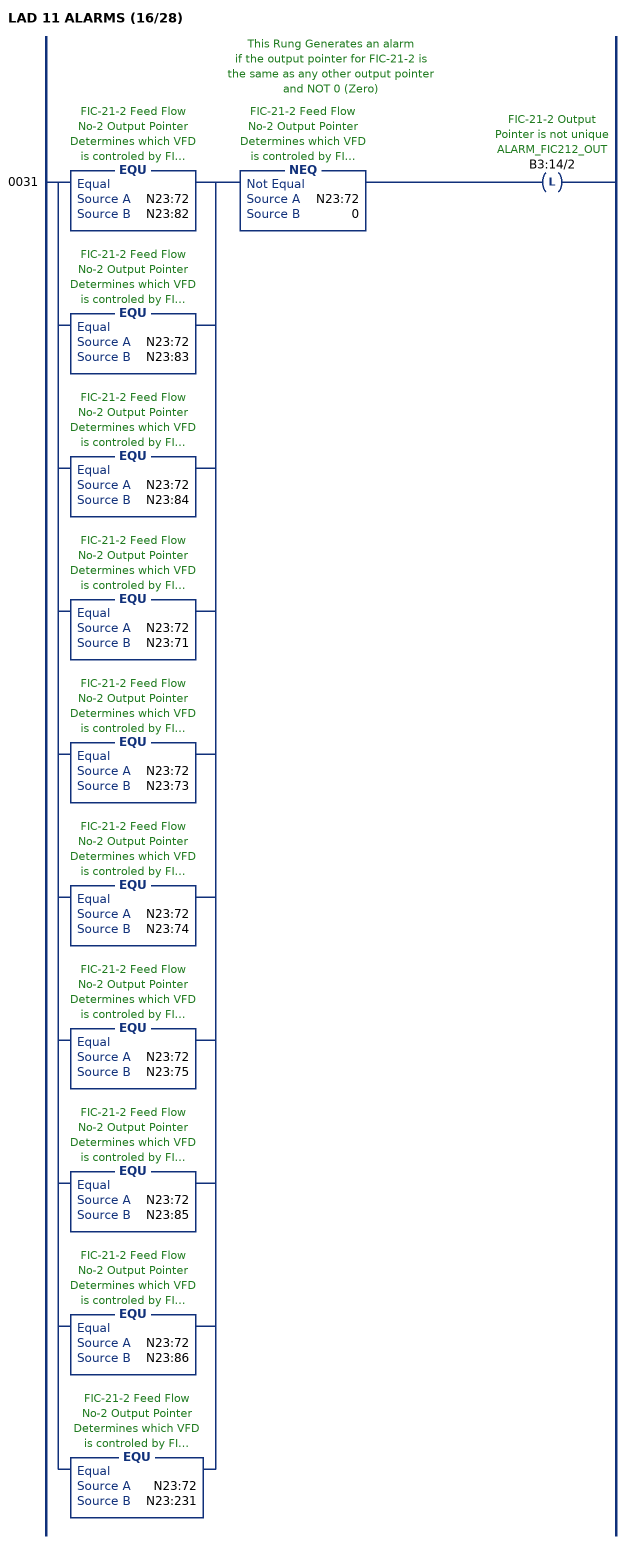
% Rung: 31 %
% This Rung Generates an alarm
% if the output pointer for FIC-21-2 is
% the same as any other output pointer
% and NOT 0 (Zero) %
SOR BST EQU N23:72 N23:82 NXB EQU N23:72 N23:83 NXB EQU N23:72 N23:84 NXB EQU N23:72 N23:71 NXB EQU N23:72 N23:73 NXB EQU N23:72 N23:74 NXB EQU N23:72 N23:75 NXB EQU N23:72 N23:85 NXB EQU N23:72 N23:86 NXB EQU N23:72 N23:231 BND NEQ N23:72 0 OTL B3:14/2 EOR
%   N23:72  FIC212_OUT_PTR  "FIC-21-2 Feed Flow No-2 Output Pointer Determines which VFD is controled by FIC" %
%   N23:82  EV02_OUT_PTR  "EV-2 Rotor Output Pointer (Selects which VFD is used by EV-2)" %
%   N23:83  EV03_OUT_PTR  "EV-3 Rotor Drive Output Pointer (Selects which VFD is used by EV-3)" %
%   N23:84  AG04_OUT_PTR  "AG-4 Agitator Output Pointer (Selects which VFD is used by AG-4)" %
%   N23:71  FIC211_OUT_PTR  "FIC-21-1 Feed Flow No-1 Output Pointer Determines which VFD is controled by FIC" %
%   N23:73  FIC213_OUT_PTR  "FIC-21-3 Feed Flow No-3 Output Pointer Determines which VFD is controled by FIC" %
%   N23:74  FIC214_OUT_PTR  "FIC-21-4 Feed Flow No-4 Output Pointer Determines which VFD is controled by FIC" %
%   N23:75  PIC461_OUT_PTR  "PIC-46-1 Flash Evap Feed Pres Output Pointer Determines which VFD is controled by FIC" %
%   N23:85  EV42_OUT_PTR  "EV-42 Rotor Drive Rotor Output Pointer (Selects which VFD is used by EV-3)" %
%   N23:86  EV20_OUT_PTR  "EV-20 Rotor Drive Rotor Output Pointer (Selects which VFD is used by EV-3)" %
%   N23:231  LIC221_OUT_PTR  "LIC-22-1 Level No-1 Output Pointer Determines which VFD is controled by LIC" %
%   B3:14/2  ALARM_FIC212_OUT  "FIC-21-2 Output Pointer is not unique" %

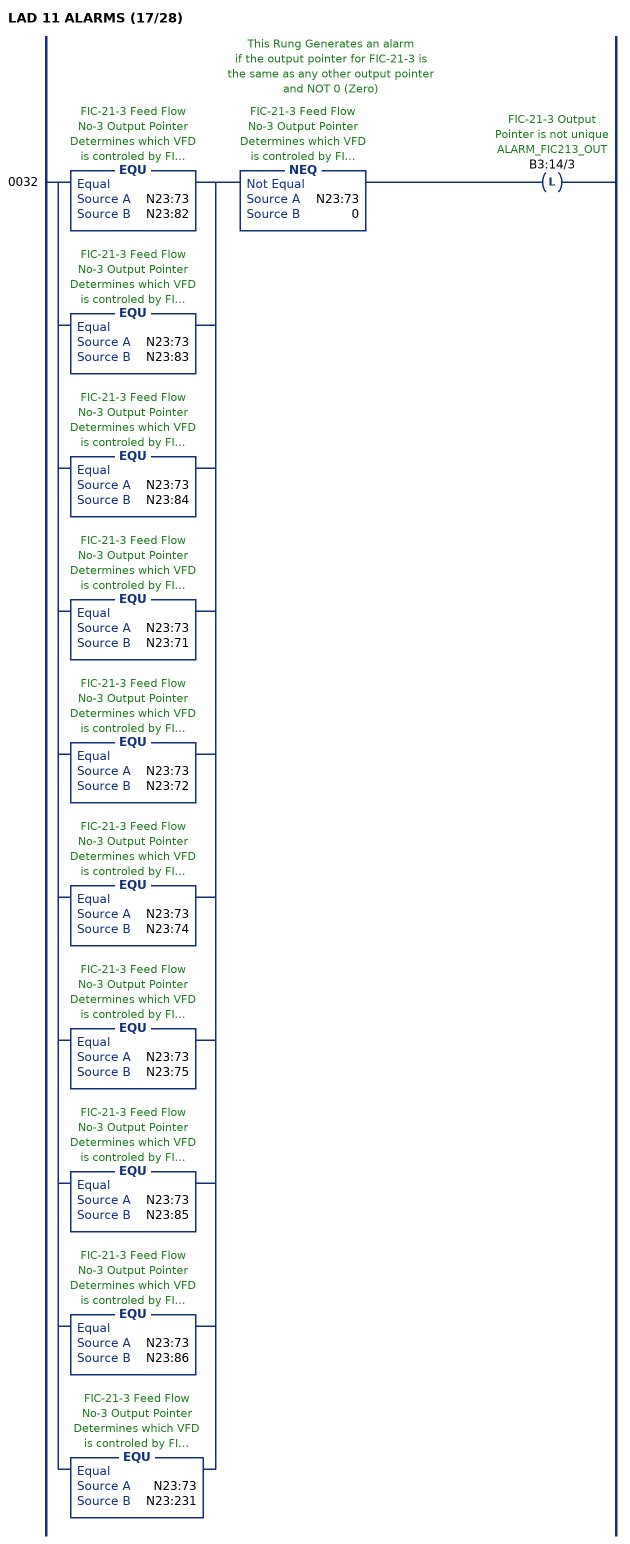
% Rung: 32 %
% This Rung Generates an alarm
% if the output pointer for FIC-21-3 is
% the same as any other output pointer
% and NOT 0 (Zero) %
SOR BST EQU N23:73 N23:82 NXB EQU N23:73 N23:83 NXB EQU N23:73 N23:84 NXB EQU N23:73 N23:71 NXB EQU N23:73 N23:72 NXB EQU N23:73 N23:74 NXB EQU N23:73 N23:75 NXB EQU N23:73 N23:85 NXB EQU N23:73 N23:86 NXB EQU N23:73 N23:231 BND NEQ N23:73 0 OTL B3:14/3 EOR
%   N23:73  FIC213_OUT_PTR  "FIC-21-3 Feed Flow No-3 Output Pointer Determines which VFD is controled by FIC" %
%   N23:82  EV02_OUT_PTR  "EV-2 Rotor Output Pointer (Selects which VFD is used by EV-2)" %
%   N23:83  EV03_OUT_PTR  "EV-3 Rotor Drive Output Pointer (Selects which VFD is used by EV-3)" %
%   N23:84  AG04_OUT_PTR  "AG-4 Agitator Output Pointer (Selects which VFD is used by AG-4)" %
%   N23:71  FIC211_OUT_PTR  "FIC-21-1 Feed Flow No-1 Output Pointer Determines which VFD is controled by FIC" %
%   N23:72  FIC212_OUT_PTR  "FIC-21-2 Feed Flow No-2 Output Pointer Determines which VFD is controled by FIC" %
%   N23:74  FIC214_OUT_PTR  "FIC-21-4 Feed Flow No-4 Output Pointer Determines which VFD is controled by FIC" %
%   N23:75  PIC461_OUT_PTR  "PIC-46-1 Flash Evap Feed Pres Output Pointer Determines which VFD is controled by FIC" %
%   N23:85  EV42_OUT_PTR  "EV-42 Rotor Drive Rotor Output Pointer (Selects which VFD is used by EV-3)" %
%   N23:86  EV20_OUT_PTR  "EV-20 Rotor Drive Rotor Output Pointer (Selects which VFD is used by EV-3)" %
%   N23:231  LIC221_OUT_PTR  "LIC-22-1 Level No-1 Output Pointer Determines which VFD is controled by LIC" %
%   B3:14/3  ALARM_FIC213_OUT  "FIC-21-3 Output Pointer is not unique" %

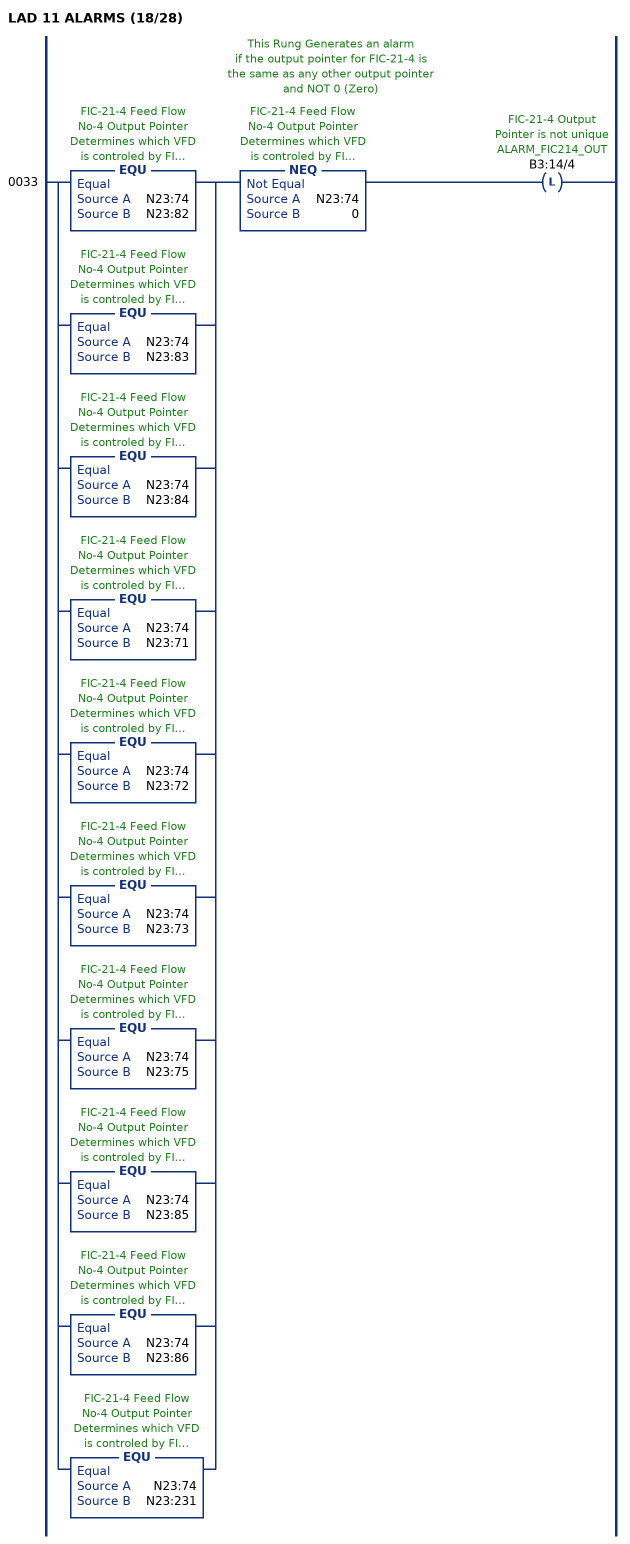
% Rung: 33 %
% This Rung Generates an alarm
% if the output pointer for FIC-21-4 is
% the same as any other output pointer
% and NOT 0 (Zero) %
SOR BST EQU N23:74 N23:82 NXB EQU N23:74 N23:83 NXB EQU N23:74 N23:84 NXB EQU N23:74 N23:71 NXB EQU N23:74 N23:72 NXB EQU N23:74 N23:73 NXB EQU N23:74 N23:75 NXB EQU N23:74 N23:85 NXB EQU N23:74 N23:86 NXB EQU N23:74 N23:231 BND NEQ N23:74 0 OTL B3:14/4 EOR
%   N23:74  FIC214_OUT_PTR  "FIC-21-4 Feed Flow No-4 Output Pointer Determines which VFD is controled by FIC" %
%   N23:82  EV02_OUT_PTR  "EV-2 Rotor Output Pointer (Selects which VFD is used by EV-2)" %
%   N23:83  EV03_OUT_PTR  "EV-3 Rotor Drive Output Pointer (Selects which VFD is used by EV-3)" %
%   N23:84  AG04_OUT_PTR  "AG-4 Agitator Output Pointer (Selects which VFD is used by AG-4)" %
%   N23:71  FIC211_OUT_PTR  "FIC-21-1 Feed Flow No-1 Output Pointer Determines which VFD is controled by FIC" %
%   N23:72  FIC212_OUT_PTR  "FIC-21-2 Feed Flow No-2 Output Pointer Determines which VFD is controled by FIC" %
%   N23:73  FIC213_OUT_PTR  "FIC-21-3 Feed Flow No-3 Output Pointer Determines which VFD is controled by FIC" %
%   N23:75  PIC461_OUT_PTR  "PIC-46-1 Flash Evap Feed Pres Output Pointer Determines which VFD is controled by FIC" %
%   N23:85  EV42_OUT_PTR  "EV-42 Rotor Drive Rotor Output Pointer (Selects which VFD is used by EV-3)" %
%   N23:86  EV20_OUT_PTR  "EV-20 Rotor Drive Rotor Output Pointer (Selects which VFD is used by EV-3)" %
%   N23:231  LIC221_OUT_PTR  "LIC-22-1 Level No-1 Output Pointer Determines which VFD is controled by LIC" %
%   B3:14/4  ALARM_FIC214_OUT  "FIC-21-4 Output Pointer is not unique" %

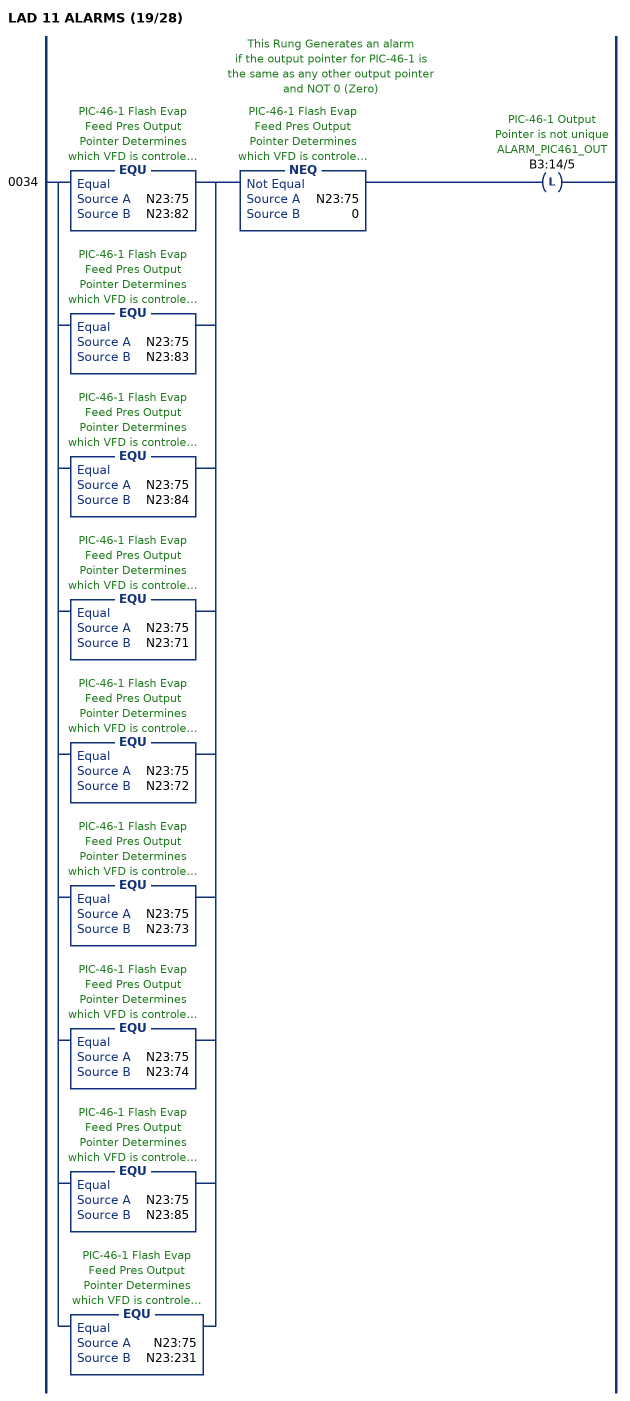
% Rung: 34 %
% This Rung Generates an alarm
% if the output pointer for PIC-46-1 is
% the same as any other output pointer
% and NOT 0 (Zero) %
SOR BST EQU N23:75 N23:82 NXB EQU N23:75 N23:83 NXB EQU N23:75 N23:84 NXB EQU N23:75 N23:71 NXB EQU N23:75 N23:72 NXB EQU N23:75 N23:73 NXB EQU N23:75 N23:74 NXB EQU N23:75 N23:85 NXB EQU N23:75 N23:231 BND NEQ N23:75 0 OTL B3:14/5 EOR
%   N23:75  PIC461_OUT_PTR  "PIC-46-1 Flash Evap Feed Pres Output Pointer Determines which VFD is controled by FIC" %
%   N23:82  EV02_OUT_PTR  "EV-2 Rotor Output Pointer (Selects which VFD is used by EV-2)" %
%   N23:83  EV03_OUT_PTR  "EV-3 Rotor Drive Output Pointer (Selects which VFD is used by EV-3)" %
%   N23:84  AG04_OUT_PTR  "AG-4 Agitator Output Pointer (Selects which VFD is used by AG-4)" %
%   N23:71  FIC211_OUT_PTR  "FIC-21-1 Feed Flow No-1 Output Pointer Determines which VFD is controled by FIC" %
%   N23:72  FIC212_OUT_PTR  "FIC-21-2 Feed Flow No-2 Output Pointer Determines which VFD is controled by FIC" %
%   N23:73  FIC213_OUT_PTR  "FIC-21-3 Feed Flow No-3 Output Pointer Determines which VFD is controled by FIC" %
%   N23:74  FIC214_OUT_PTR  "FIC-21-4 Feed Flow No-4 Output Pointer Determines which VFD is controled by FIC" %
%   N23:85  EV42_OUT_PTR  "EV-42 Rotor Drive Rotor Output Pointer (Selects which VFD is used by EV-3)" %
%   N23:231  LIC221_OUT_PTR  "LIC-22-1 Level No-1 Output Pointer Determines which VFD is controled by LIC" %
%   B3:14/5  ALARM_PIC461_OUT  "PIC-46-1 Output Pointer is not unique" %

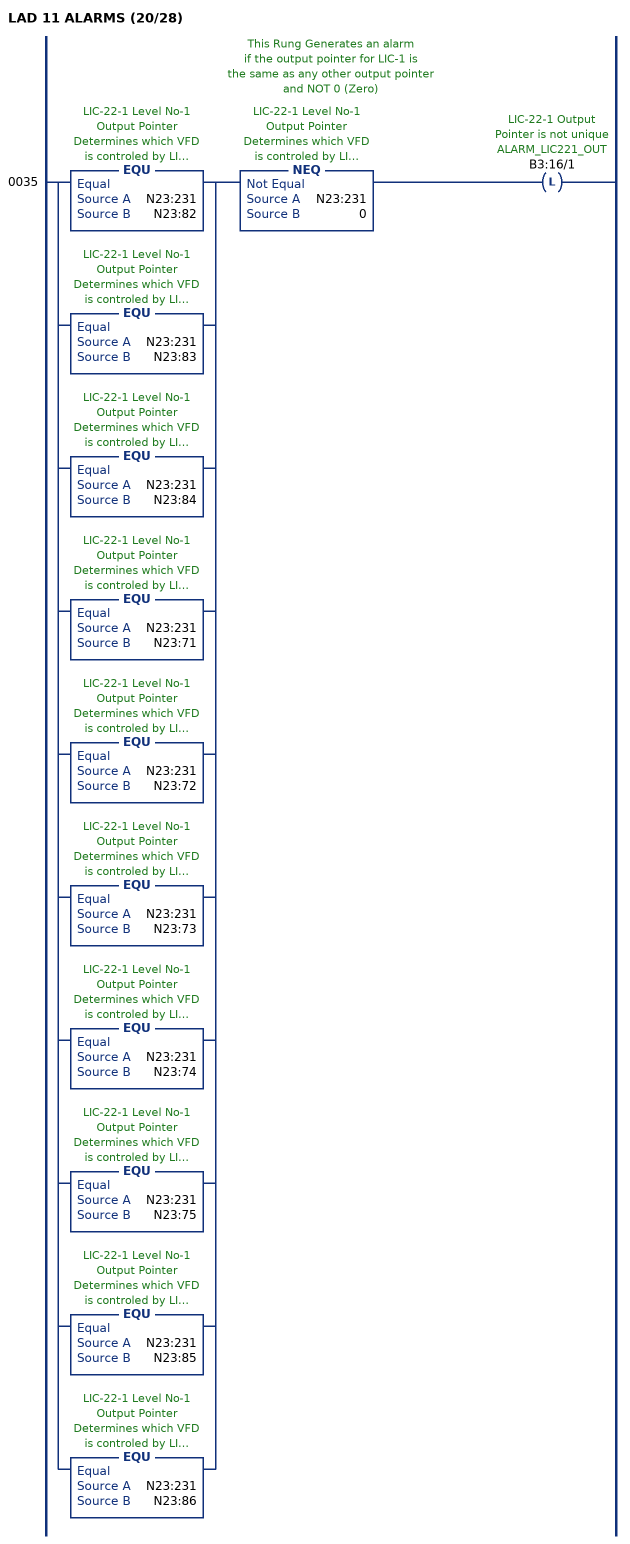
% Rung: 35 %
% This Rung Generates an alarm
% if the output pointer for LIC-1 is
% the same as any other output pointer
% and NOT 0 (Zero) %
SOR BST EQU N23:231 N23:82 NXB EQU N23:231 N23:83 NXB EQU N23:231 N23:84 NXB EQU N23:231 N23:71 NXB EQU N23:231 N23:72 NXB EQU N23:231 N23:73 NXB EQU N23:231 N23:74 NXB EQU N23:231 N23:75 NXB EQU N23:231 N23:85 NXB EQU N23:231 N23:86 BND NEQ N23:231 0 OTL B3:16/1 EOR
%   N23:231  LIC221_OUT_PTR  "LIC-22-1 Level No-1 Output Pointer Determines which VFD is controled by LIC" %
%   N23:82  EV02_OUT_PTR  "EV-2 Rotor Output Pointer (Selects which VFD is used by EV-2)" %
%   N23:83  EV03_OUT_PTR  "EV-3 Rotor Drive Output Pointer (Selects which VFD is used by EV-3)" %
%   N23:84  AG04_OUT_PTR  "AG-4 Agitator Output Pointer (Selects which VFD is used by AG-4)" %
%   N23:71  FIC211_OUT_PTR  "FIC-21-1 Feed Flow No-1 Output Pointer Determines which VFD is controled by FIC" %
%   N23:72  FIC212_OUT_PTR  "FIC-21-2 Feed Flow No-2 Output Pointer Determines which VFD is controled by FIC" %
%   N23:73  FIC213_OUT_PTR  "FIC-21-3 Feed Flow No-3 Output Pointer Determines which VFD is controled by FIC" %
%   N23:74  FIC214_OUT_PTR  "FIC-21-4 Feed Flow No-4 Output Pointer Determines which VFD is controled by FIC" %
%   N23:75  PIC461_OUT_PTR  "PIC-46-1 Flash Evap Feed Pres Output Pointer Determines which VFD is controled by FIC" %
%   N23:85  EV42_OUT_PTR  "EV-42 Rotor Drive Rotor Output Pointer (Selects which VFD is used by EV-3)" %
%   N23:86  EV20_OUT_PTR  "EV-20 Rotor Drive Rotor Output Pointer (Selects which VFD is used by EV-3)" %
%   B3:16/1  ALARM_LIC221_OUT  "LIC-22-1 Output Pointer is not unique" %

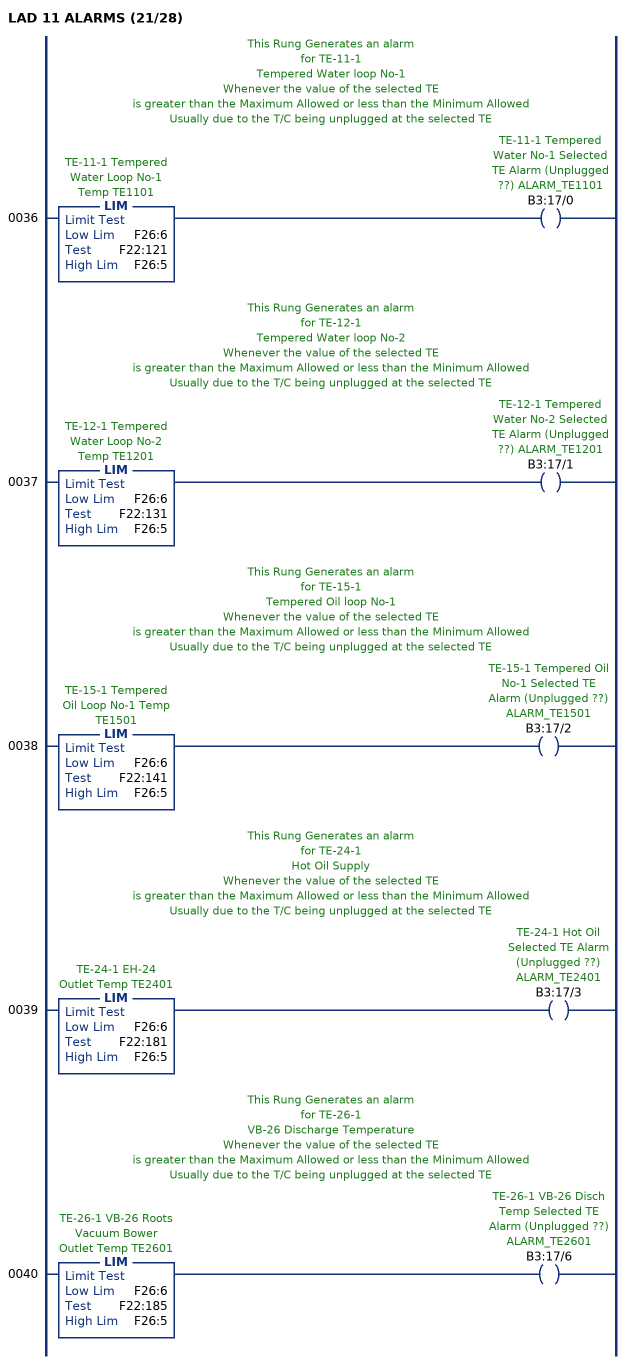
% Rung: 36 %
% This Rung Generates an alarm
% for TE-11-1
% Tempered Water loop No-1
% Whenever the value of the selected TE
% is greater than the Maximum Allowed or less than the Minimum Allowed
% Usually due to the T/C being unplugged at the selected TE %
SOR LIM F26:6 F22:121 F26:5 OTE B3:17/0 EOR
%   F26:6  TE_MAX  "TE Input Maximum Value if TE is >= this value an alarm is generated" %
%   F22:121  TE1101  "TE-11-1 Tempered Water Loop No-1 Temp" %
%   F26:5  TE_MIN  "TE Input Minimum Value if TE is <= this value an alarm is generated" %
%   B3:17/0  ALARM_TE1101  "TE-11-1 Tempered Water No-1 Selected TE Alarm (Unplugged ??)" %
% Rung: 37 %
% This Rung Generates an alarm
% for TE-12-1
% Tempered Water loop No-2
% Whenever the value of the selected TE
% is greater than the Maximum Allowed or less than the Minimum Allowed
% Usually due to the T/C being unplugged at the selected TE %
SOR LIM F26:6 F22:131 F26:5 OTE B3:17/1 EOR
%   F26:6  TE_MAX  "TE Input Maximum Value if TE is >= this value an alarm is generated" %
%   F22:131  TE1201  "TE-12-1 Tempered Water Loop No-2 Temp" %
%   F26:5  TE_MIN  "TE Input Minimum Value if TE is <= this value an alarm is generated" %
%   B3:17/1  ALARM_TE1201  "TE-12-1 Tempered Water No-2 Selected TE Alarm (Unplugged ??)" %
% Rung: 38 %
% This Rung Generates an alarm
% for TE-15-1
% Tempered Oil loop No-1
% Whenever the value of the selected TE
% is greater than the Maximum Allowed or less than the Minimum Allowed
% Usually due to the T/C being unplugged at the selected TE %
SOR LIM F26:6 F22:141 F26:5 OTE B3:17/2 EOR
%   F26:6  TE_MAX  "TE Input Maximum Value if TE is >= this value an alarm is generated" %
%   F22:141  TE1501  "TE-15-1 Tempered Oil Loop No-1 Temp" %
%   F26:5  TE_MIN  "TE Input Minimum Value if TE is <= this value an alarm is generated" %
%   B3:17/2  ALARM_TE1501  "TE-15-1 Tempered Oil No-1 Selected TE Alarm (Unplugged ??)" %
% Rung: 39 %
% This Rung Generates an alarm
% for TE-24-1
% Hot Oil Supply
% Whenever the value of the selected TE
% is greater than the Maximum Allowed or less than the Minimum Allowed
% Usually due to the T/C being unplugged at the selected TE %
SOR LIM F26:6 F22:181 F26:5 OTE B3:17/3 EOR
%   F26:6  TE_MAX  "TE Input Maximum Value if TE is >= this value an alarm is generated" %
%   F22:181  TE2401  "TE-24-1 EH-24 Outlet Temp" %
%   F26:5  TE_MIN  "TE Input Minimum Value if TE is <= this value an alarm is generated" %
%   B3:17/3  ALARM_TE2401  "TE-24-1 Hot Oil Selected TE Alarm (Unplugged ??)" %
% Rung: 40 %
% This Rung Generates an alarm
% for TE-26-1
% VB-26 Discharge Temperature
% Whenever the value of the selected TE
% is greater than the Maximum Allowed or less than the Minimum Allowed
% Usually due to the T/C being unplugged at the selected TE %
SOR LIM F26:6 F22:185 F26:5 OTE B3:17/6 EOR
%   F26:6  TE_MAX  "TE Input Maximum Value if TE is >= this value an alarm is generated" %
%   F22:185  TE2601  "TE-26-1 VB-26 Roots Vacuum Bower Outlet Temp" %
%   F26:5  TE_MIN  "TE Input Minimum Value if TE is <= this value an alarm is generated" %
%   B3:17/6  ALARM_TE2601  "TE-26-1 VB-26 Disch Temp Selected TE Alarm (Unplugged ??)" %

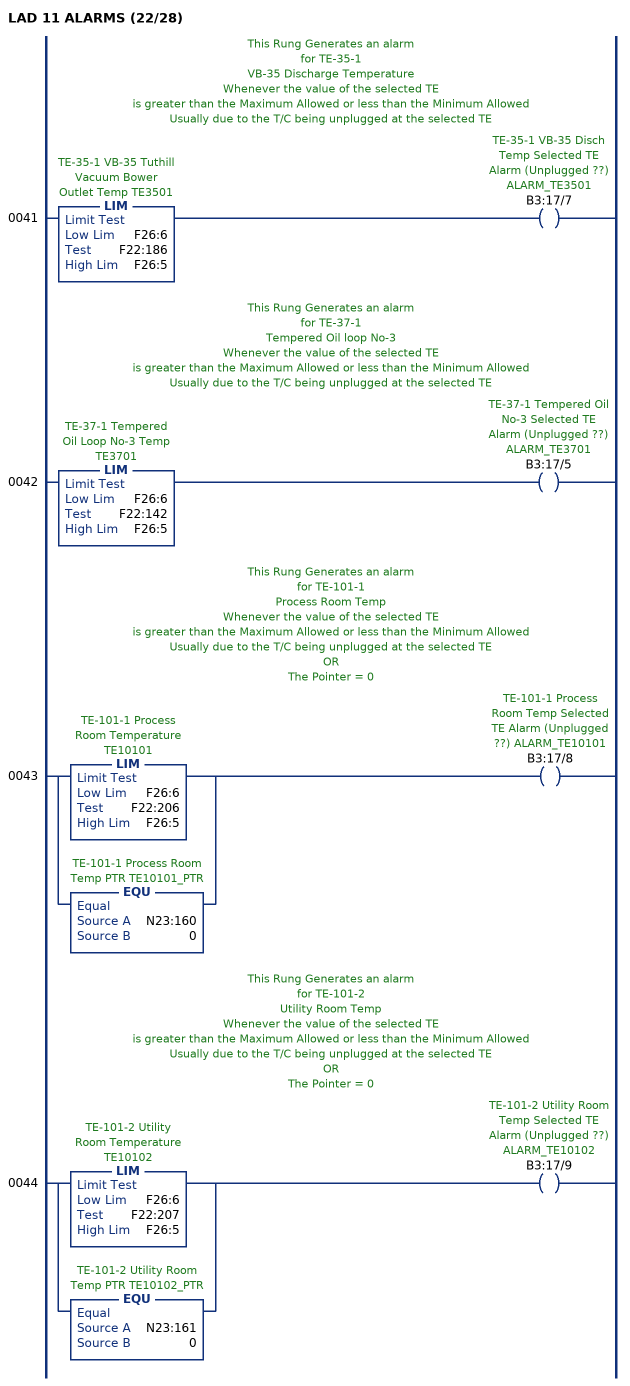
% Rung: 41 %
% This Rung Generates an alarm
% for TE-35-1
% VB-35 Discharge Temperature
% Whenever the value of the selected TE
% is greater than the Maximum Allowed or less than the Minimum Allowed
% Usually due to the T/C being unplugged at the selected TE %
SOR LIM F26:6 F22:186 F26:5 OTE B3:17/7 EOR
%   F26:6  TE_MAX  "TE Input Maximum Value if TE is >= this value an alarm is generated" %
%   F22:186  TE3501  "TE-35-1 VB-35 Tuthill Vacuum Bower Outlet Temp" %
%   F26:5  TE_MIN  "TE Input Minimum Value if TE is <= this value an alarm is generated" %
%   B3:17/7  ALARM_TE3501  "TE-35-1 VB-35 Disch Temp Selected TE Alarm (Unplugged ??)" %
% Rung: 42 %
% This Rung Generates an alarm
% for TE-37-1
% Tempered Oil loop No-3
% Whenever the value of the selected TE
% is greater than the Maximum Allowed or less than the Minimum Allowed
% Usually due to the T/C being unplugged at the selected TE %
SOR LIM F26:6 F22:142 F26:5 OTE B3:17/5 EOR
%   F26:6  TE_MAX  "TE Input Maximum Value if TE is >= this value an alarm is generated" %
%   F22:142  TE3701  "TE-37-1 Tempered Oil Loop No-3 Temp" %
%   F26:5  TE_MIN  "TE Input Minimum Value if TE is <= this value an alarm is generated" %
%   B3:17/5  ALARM_TE3701  "TE-37-1 Tempered Oil No-3 Selected TE Alarm (Unplugged ??)" %
% Rung: 43 %
% This Rung Generates an alarm
% for TE-101-1
% Process Room Temp
% Whenever the value of the selected TE
% is greater than the Maximum Allowed or less than the Minimum Allowed
% Usually due to the T/C being unplugged at the selected TE
% OR
% The Pointer = 0 %
SOR BST LIM F26:6 F22:206 F26:5 NXB EQU N23:160 0 BND OTE B3:17/8 EOR
%   F26:6  TE_MAX  "TE Input Maximum Value if TE is >= this value an alarm is generated" %
%   F22:206  TE10101  "TE-101-1 Process Room Temperature" %
%   F26:5  TE_MIN  "TE Input Minimum Value if TE is <= this value an alarm is generated" %
%   N23:160  TE10101_PTR  "TE-101-1 Process Room Temp PTR" %
%   B3:17/8  ALARM_TE10101  "TE-101-1 Process Room Temp Selected TE Alarm (Unplugged ??)" %
% Rung: 44 %
% This Rung Generates an alarm
% for TE-101-2
% Utility Room Temp
% Whenever the value of the selected TE
% is greater than the Maximum Allowed or less than the Minimum Allowed
% Usually due to the T/C being unplugged at the selected TE
% OR
% The Pointer = 0 %
SOR BST LIM F26:6 F22:207 F26:5 NXB EQU N23:161 0 BND OTE B3:17/9 EOR
%   F26:6  TE_MAX  "TE Input Maximum Value if TE is >= this value an alarm is generated" %
%   F22:207  TE10102  "TE-101-2 Utility Room Temperature" %
%   F26:5  TE_MIN  "TE Input Minimum Value if TE is <= this value an alarm is generated" %
%   N23:161  TE10102_PTR  "TE-101-2 Utility Room Temp PTR" %
%   B3:17/9  ALARM_TE10102  "TE-101-2 Utility Room Temp Selected TE Alarm (Unplugged ??)" %

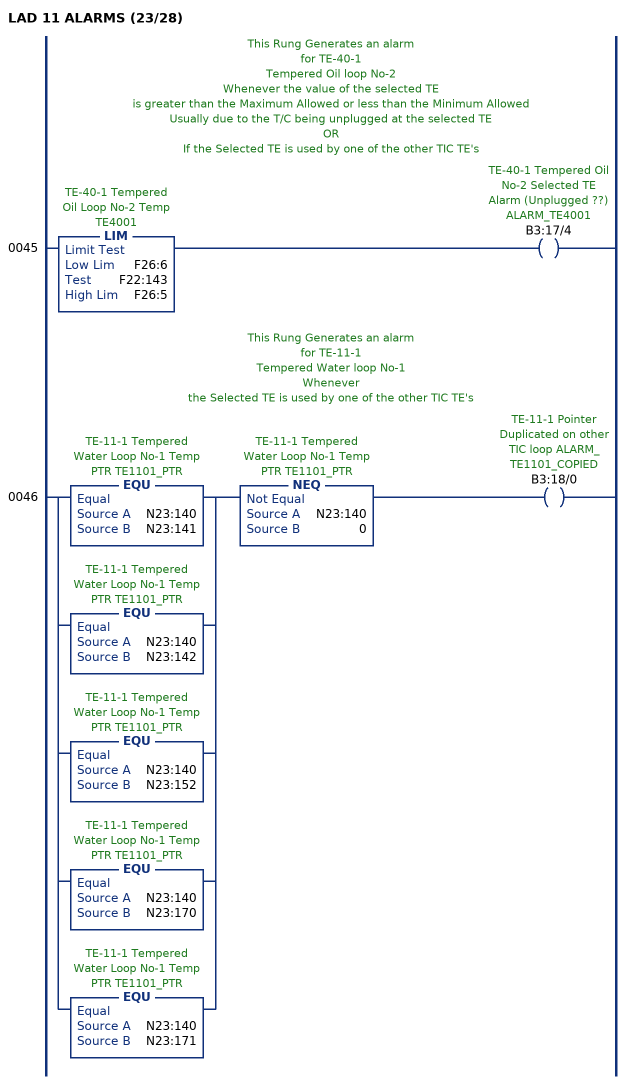
% Rung: 45 %
% This Rung Generates an alarm
% for TE-40-1
% Tempered Oil loop No-2
% Whenever the value of the selected TE
% is greater than the Maximum Allowed or less than the Minimum Allowed
% Usually due to the T/C being unplugged at the selected TE
% OR
% If the Selected TE is used by one of the other TIC TE's %
SOR LIM F26:6 F22:143 F26:5 OTE B3:17/4 EOR
%   F26:6  TE_MAX  "TE Input Maximum Value if TE is >= this value an alarm is generated" %
%   F22:143  TE4001  "TE-40-1 Tempered Oil Loop No-2 Temp" %
%   F26:5  TE_MIN  "TE Input Minimum Value if TE is <= this value an alarm is generated" %
%   B3:17/4  ALARM_TE4001  "TE-40-1 Tempered Oil No-2 Selected TE Alarm (Unplugged ??)" %
% Rung: 46 %
% This Rung Generates an alarm
% for TE-11-1
% Tempered Water loop No-1
% Whenever
% the Selected TE is used by one of the other TIC TE's %
SOR BST EQU N23:140 N23:141 NXB EQU N23:140 N23:142 NXB EQU N23:140 N23:152 NXB EQU N23:140 N23:170 NXB EQU N23:140 N23:171 BND NEQ N23:140 0 OTE B3:18/0 EOR
%   N23:140  TE1101_PTR  "TE-11-1 Tempered Water Loop No-1 Temp PTR" %
%   N23:141  TE1201_PTR  "TE-12-1 Tempered Water Loop No-2 Temp PTR" %
%   N23:142  TE1501_PTR  "TE-15-1 Tempered Oil Loop No-1 Temp PTR" %
%   N23:152  TE2401_PTR  "TE-24-1 EH-24 Outlet Temp PTR" %
%   N23:170  TE3701_PTR  "TE-37-1 Tempered Oil Loop No-3 Temp PTR" %
%   N23:171  TE4001_PTR  "TE-40-1 Tempered Oil Loop No-2 Temp PTR" %
%   B3:18/0  ALARM_TE1101_COPIED  "TE-11-1 Pointer Duplicated on other TIC loop" %

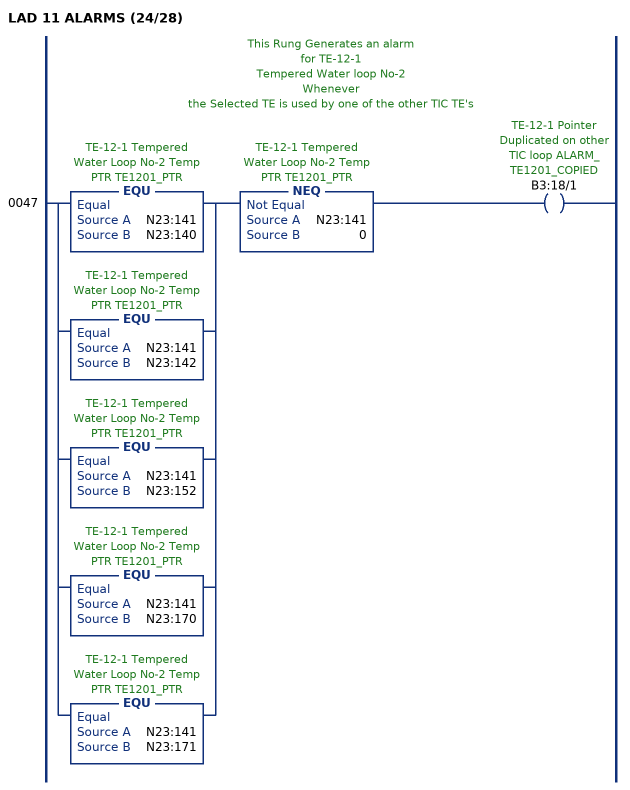
% Rung: 47 %
% This Rung Generates an alarm
% for TE-12-1
% Tempered Water loop No-2
% Whenever
% the Selected TE is used by one of the other TIC TE's %
SOR BST EQU N23:141 N23:140 NXB EQU N23:141 N23:142 NXB EQU N23:141 N23:152 NXB EQU N23:141 N23:170 NXB EQU N23:141 N23:171 BND NEQ N23:141 0 OTE B3:18/1 EOR
%   N23:141  TE1201_PTR  "TE-12-1 Tempered Water Loop No-2 Temp PTR" %
%   N23:140  TE1101_PTR  "TE-11-1 Tempered Water Loop No-1 Temp PTR" %
%   N23:142  TE1501_PTR  "TE-15-1 Tempered Oil Loop No-1 Temp PTR" %
%   N23:152  TE2401_PTR  "TE-24-1 EH-24 Outlet Temp PTR" %
%   N23:170  TE3701_PTR  "TE-37-1 Tempered Oil Loop No-3 Temp PTR" %
%   N23:171  TE4001_PTR  "TE-40-1 Tempered Oil Loop No-2 Temp PTR" %
%   B3:18/1  ALARM_TE1201_COPIED  "TE-12-1 Pointer Duplicated on other TIC loop" %

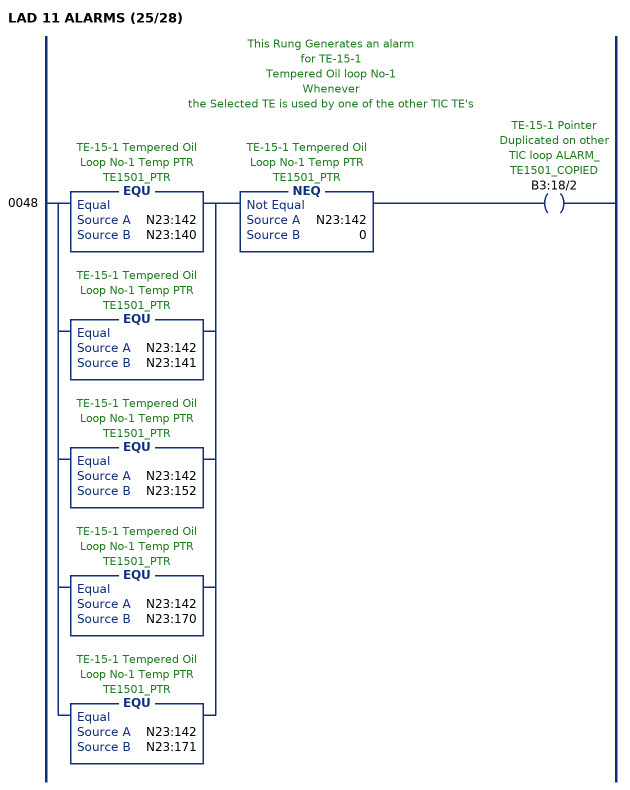
% Rung: 48 %
% This Rung Generates an alarm
% for TE-15-1
% Tempered Oil loop No-1
% Whenever
% the Selected TE is used by one of the other TIC TE's %
SOR BST EQU N23:142 N23:140 NXB EQU N23:142 N23:141 NXB EQU N23:142 N23:152 NXB EQU N23:142 N23:170 NXB EQU N23:142 N23:171 BND NEQ N23:142 0 OTE B3:18/2 EOR
%   N23:142  TE1501_PTR  "TE-15-1 Tempered Oil Loop No-1 Temp PTR" %
%   N23:140  TE1101_PTR  "TE-11-1 Tempered Water Loop No-1 Temp PTR" %
%   N23:141  TE1201_PTR  "TE-12-1 Tempered Water Loop No-2 Temp PTR" %
%   N23:152  TE2401_PTR  "TE-24-1 EH-24 Outlet Temp PTR" %
%   N23:170  TE3701_PTR  "TE-37-1 Tempered Oil Loop No-3 Temp PTR" %
%   N23:171  TE4001_PTR  "TE-40-1 Tempered Oil Loop No-2 Temp PTR" %
%   B3:18/2  ALARM_TE1501_COPIED  "TE-15-1 Pointer Duplicated on other TIC loop" %

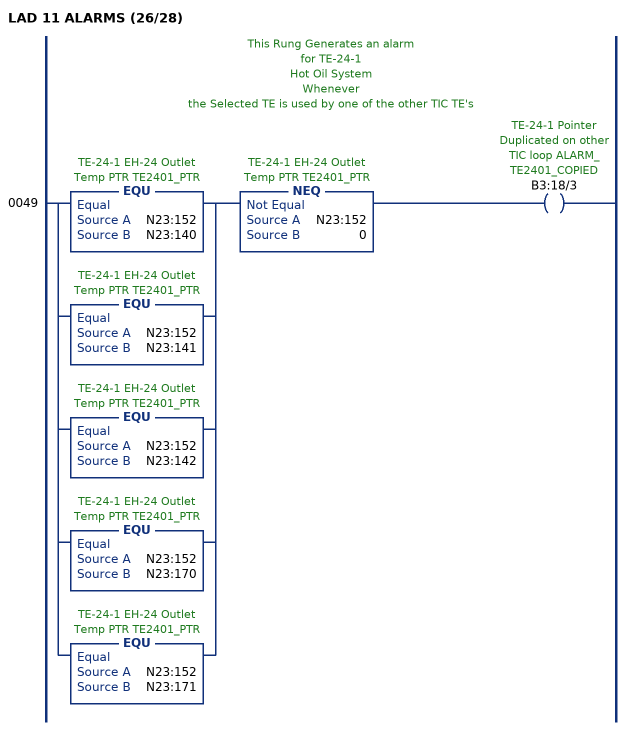
% Rung: 49 %
% This Rung Generates an alarm
% for TE-24-1
% Hot Oil System
% Whenever
% the Selected TE is used by one of the other TIC TE's %
SOR BST EQU N23:152 N23:140 NXB EQU N23:152 N23:141 NXB EQU N23:152 N23:142 NXB EQU N23:152 N23:170 NXB EQU N23:152 N23:171 BND NEQ N23:152 0 OTE B3:18/3 EOR
%   N23:152  TE2401_PTR  "TE-24-1 EH-24 Outlet Temp PTR" %
%   N23:140  TE1101_PTR  "TE-11-1 Tempered Water Loop No-1 Temp PTR" %
%   N23:141  TE1201_PTR  "TE-12-1 Tempered Water Loop No-2 Temp PTR" %
%   N23:142  TE1501_PTR  "TE-15-1 Tempered Oil Loop No-1 Temp PTR" %
%   N23:170  TE3701_PTR  "TE-37-1 Tempered Oil Loop No-3 Temp PTR" %
%   N23:171  TE4001_PTR  "TE-40-1 Tempered Oil Loop No-2 Temp PTR" %
%   B3:18/3  ALARM_TE2401_COPIED  "TE-24-1 Pointer Duplicated on other TIC loop" %

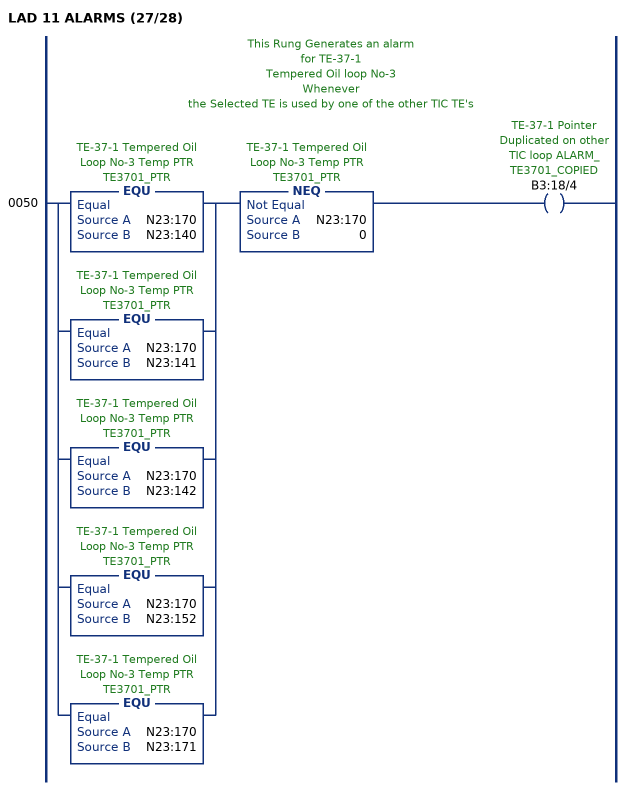
% Rung: 50 %
% This Rung Generates an alarm
% for TE-37-1
% Tempered Oil loop No-3
% Whenever
% the Selected TE is used by one of the other TIC TE's %
SOR BST EQU N23:170 N23:140 NXB EQU N23:170 N23:141 NXB EQU N23:170 N23:142 NXB EQU N23:170 N23:152 NXB EQU N23:170 N23:171 BND NEQ N23:170 0 OTE B3:18/4 EOR
%   N23:170  TE3701_PTR  "TE-37-1 Tempered Oil Loop No-3 Temp PTR" %
%   N23:140  TE1101_PTR  "TE-11-1 Tempered Water Loop No-1 Temp PTR" %
%   N23:141  TE1201_PTR  "TE-12-1 Tempered Water Loop No-2 Temp PTR" %
%   N23:142  TE1501_PTR  "TE-15-1 Tempered Oil Loop No-1 Temp PTR" %
%   N23:152  TE2401_PTR  "TE-24-1 EH-24 Outlet Temp PTR" %
%   N23:171  TE4001_PTR  "TE-40-1 Tempered Oil Loop No-2 Temp PTR" %
%   B3:18/4  ALARM_TE3701_COPIED  "TE-37-1 Pointer Duplicated on other TIC loop" %

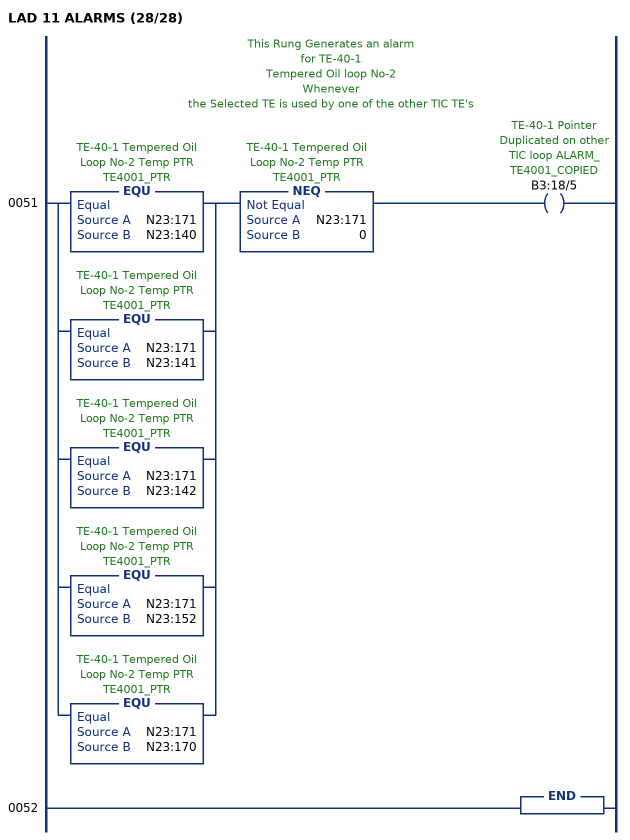
% Rung: 51 %
% This Rung Generates an alarm
% for TE-40-1
% Tempered Oil loop No-2
% Whenever
% the Selected TE is used by one of the other TIC TE's %
SOR BST EQU N23:171 N23:140 NXB EQU N23:171 N23:141 NXB EQU N23:171 N23:142 NXB EQU N23:171 N23:152 NXB EQU N23:171 N23:170 BND NEQ N23:171 0 OTE B3:18/5 EOR
%   N23:171  TE4001_PTR  "TE-40-1 Tempered Oil Loop No-2 Temp PTR" %
%   N23:140  TE1101_PTR  "TE-11-1 Tempered Water Loop No-1 Temp PTR" %
%   N23:141  TE1201_PTR  "TE-12-1 Tempered Water Loop No-2 Temp PTR" %
%   N23:142  TE1501_PTR  "TE-15-1 Tempered Oil Loop No-1 Temp PTR" %
%   N23:152  TE2401_PTR  "TE-24-1 EH-24 Outlet Temp PTR" %
%   N23:170  TE3701_PTR  "TE-37-1 Tempered Oil Loop No-3 Temp PTR" %
%   B3:18/5  ALARM_TE4001_COPIED  "TE-40-1 Pointer Duplicated on other TIC loop" %
% Rung: 52 %
SOR END EOR

LADDER 15 "IFIX PBS"    % iFIX PBs %
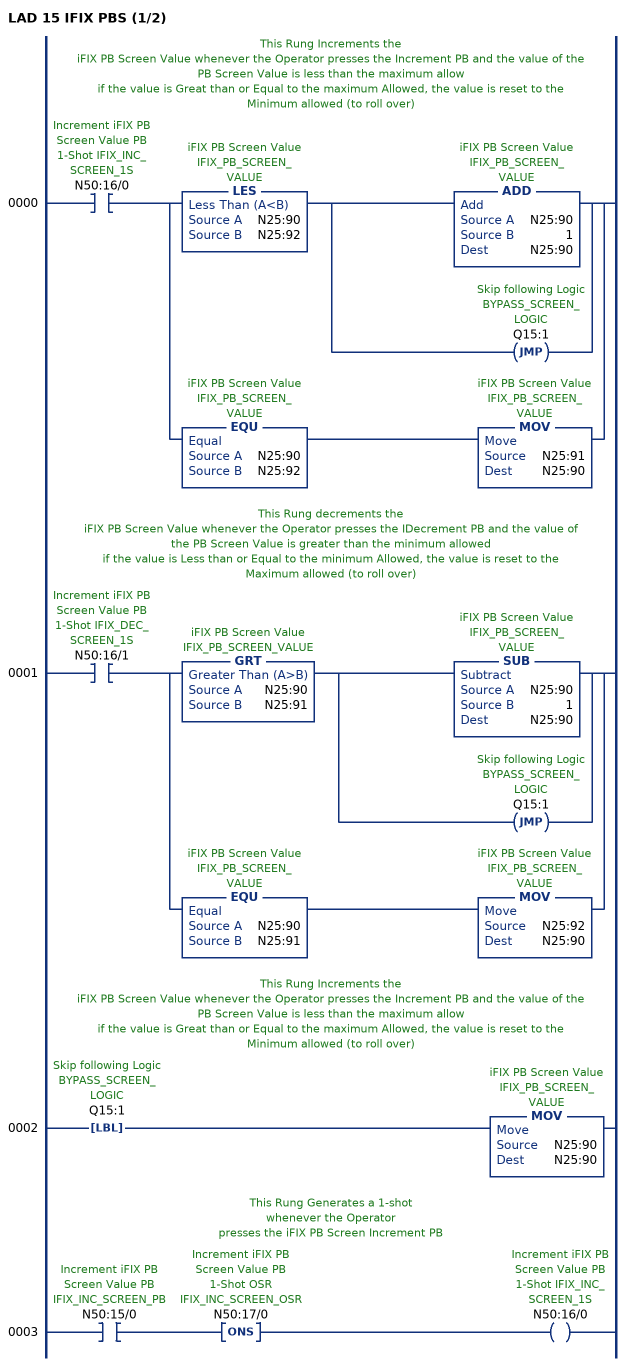
% Rung: 0 %
% This Rung Increments the
% iFIX PB Screen Value whenever the Operator presses the Increment PB and the value of the PB Screen Value is less than the maximum allow
% if the value is Great than or Equal to the maximum Allowed, the value is reset to the Minimum allowed (to roll over) %
SOR XIC N50:16/0 BST LES N25:90 N25:92 BST ADD N25:90 1 N25:90 NXB JMP Q15:1 BND NXB EQU N25:90 N25:92 MOV N25:91 N25:90 BND EOR
%   N50:16/0  IFIX_INC_SCREEN_1S  "Increment iFIX PB Screen Value PB 1-Shot" %
%   N25:90  IFIX_PB_SCREEN_VALUE  "iFIX PB Screen Value" %
%   N25:92  IFIX_PB_SCREEN_MAX  "iFIX PB Screen Minimum Value" %
%   Q15:1  BYPASS_SCREEN_LOGIC  "Skip following Logic" %
%   N25:91  IFIX_PB_SCREEN_MIN  "iFIX PB Screen Maximum Value" %
% Rung: 1 %
% This Rung decrements the
% iFIX PB Screen Value whenever the Operator presses the IDecrement PB and the value of the PB Screen Value is greater than the minimum allowed
% if the value is Less than or Equal to the minimum Allowed, the value is reset to the Maximum allowed (to roll over) %
SOR XIC N50:16/1 BST GRT N25:90 N25:91 BST SUB N25:90 1 N25:90 NXB JMP Q15:1 BND NXB EQU N25:90 N25:91 MOV N25:92 N25:90 BND EOR
%   N50:16/1  IFIX_DEC_SCREEN_1S  "Increment iFIX PB Screen Value PB 1-Shot" %
%   N25:90  IFIX_PB_SCREEN_VALUE  "iFIX PB Screen Value" %
%   N25:91  IFIX_PB_SCREEN_MIN  "iFIX PB Screen Maximum Value" %
%   Q15:1  BYPASS_SCREEN_LOGIC  "Skip following Logic" %
%   N25:92  IFIX_PB_SCREEN_MAX  "iFIX PB Screen Minimum Value" %
% Rung: 2 %
% This Rung Increments the
% iFIX PB Screen Value whenever the Operator presses the Increment PB and the value of the PB Screen Value is less than the maximum allow
% if the value is Great than or Equal to the maximum Allowed, the value is reset to the Minimum allowed (to roll over) %
SOR LBL Q15:1 MOV N25:90 N25:90 EOR
%   Q15:1  BYPASS_SCREEN_LOGIC  "Skip following Logic" %
%   N25:90  IFIX_PB_SCREEN_VALUE  "iFIX PB Screen Value" %
% Rung: 3 %
% This Rung Generates a 1-shot
% whenever the Operator
% presses the iFIX PB Screen Increment PB %
SOR XIC N50:15/0 OSR N50:17/0 OTE N50:16/0 EOR
%   N50:15/0  IFIX_INC_SCREEN_PB  "Increment iFIX PB Screen Value PB" %
%   N50:17/0  IFIX_INC_SCREEN_OSR  "Increment iFIX PB Screen Value PB 1-Shot OSR" %
%   N50:16/0  IFIX_INC_SCREEN_1S  "Increment iFIX PB Screen Value PB 1-Shot" %

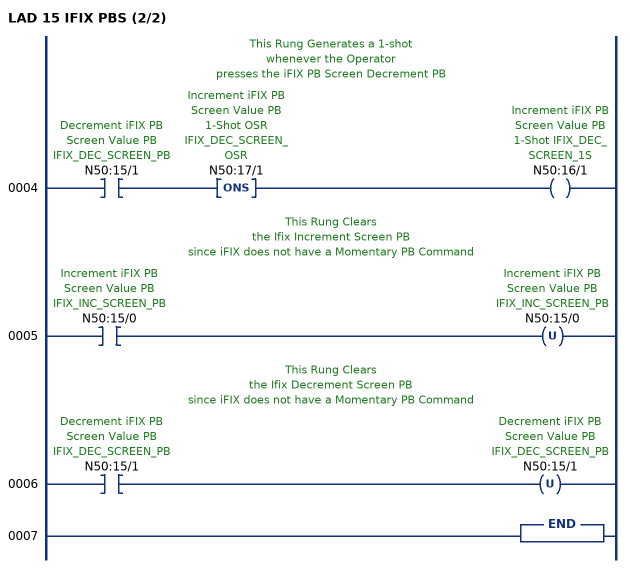
% Rung: 4 %
% This Rung Generates a 1-shot
% whenever the Operator
% presses the iFIX PB Screen Decrement PB %
SOR XIC N50:15/1 OSR N50:17/1 OTE N50:16/1 EOR
%   N50:15/1  IFIX_DEC_SCREEN_PB  "Decrement iFIX PB Screen Value PB" %
%   N50:17/1  IFIX_DEC_SCREEN_OSR  "Increment iFIX PB Screen Value PB 1-Shot OSR" %
%   N50:16/1  IFIX_DEC_SCREEN_1S  "Increment iFIX PB Screen Value PB 1-Shot" %
% Rung: 5 %
% This Rung Clears
% the Ifix Increment Screen PB
% since iFIX does not have a Momentary PB Command %
SOR XIC N50:15/0 OTU N50:15/0 EOR
%   N50:15/0  IFIX_INC_SCREEN_PB  "Increment iFIX PB Screen Value PB" %
% Rung: 6 %
% This Rung Clears
% the Ifix Decrement Screen PB
% since iFIX does not have a Momentary PB Command %
SOR XIC N50:15/1 OTU N50:15/1 EOR
%   N50:15/1  IFIX_DEC_SCREEN_PB  "Decrement iFIX PB Screen Value PB" %
% Rung: 7 %
SOR END EOR

LADDER 16 "PV PBS"    % Panel View Screen Movement PB's %
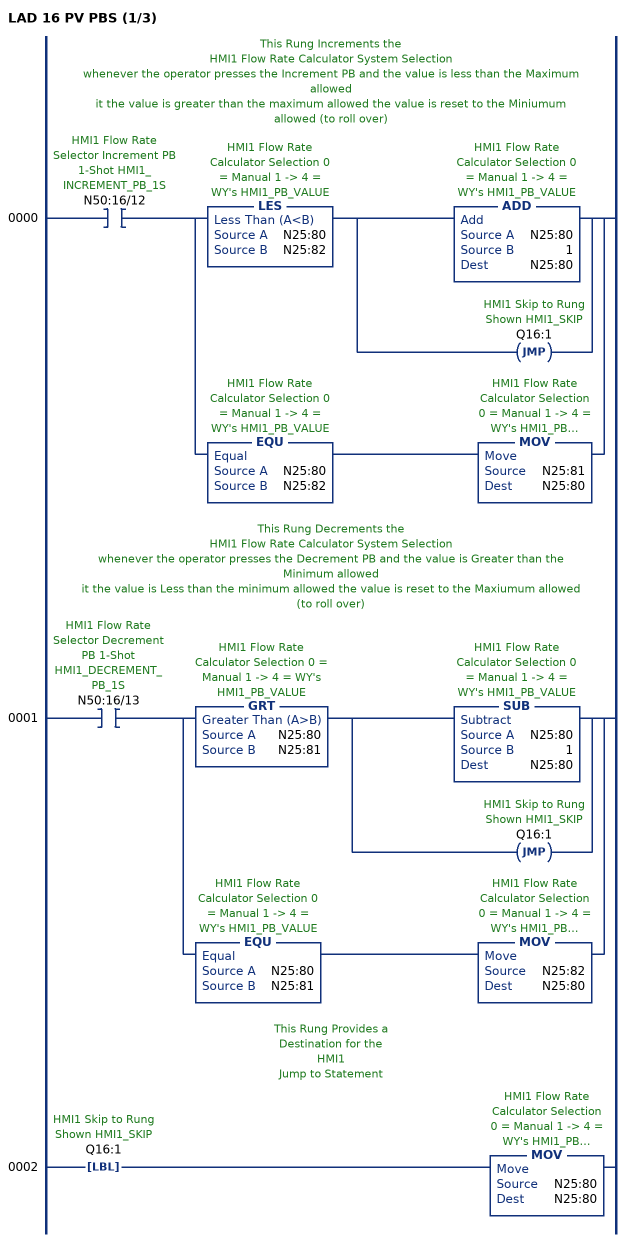
% Rung: 0 %
% This Rung Increments the
% HMI1 Flow Rate Calculator System Selection
% whenever the operator presses the Increment PB and the value is less than the Maximum allowed
% it the value is greater than the maximum allowed the value is reset to the Miniumum allowed (to roll over) %
SOR XIC N50:16/12 BST LES N25:80 N25:82 BST ADD N25:80 1 N25:80 NXB JMP Q16:1 BND NXB EQU N25:80 N25:82 MOV N25:81 N25:80 BND EOR
%   N50:16/12  HMI1_INCREMENT_PB_1S  "HMI1 Flow Rate Selector Increment PB 1-Shot" %
%   N25:80  HMI1_PB_VALUE  "HMI1 Flow Rate Calculator Selection 0 = Manual 1 -> 4 = WY's" %
%   N25:82  HMI_PB_MAX  "HMI Flow Rate Calculator Selection Maximum Value -4" %
%   Q16:1  HMI1_SKIP  "HMI1 Skip to Rung Shown" %
%   N25:81  HMI_PB_MIN  "HMI Flow Rate Calculator Selection Minimum Value 0" %
% Rung: 1 %
% This Rung Decrements the
% HMI1 Flow Rate Calculator System Selection
% whenever the operator presses the Decrement PB and the value is Greater than the Minimum allowed
% it the value is Less than the minimum allowed the value is reset to the Maxiumum allowed (to roll over) %
SOR XIC N50:16/13 BST GRT N25:80 N25:81 BST SUB N25:80 1 N25:80 NXB JMP Q16:1 BND NXB EQU N25:80 N25:81 MOV N25:82 N25:80 BND EOR
%   N50:16/13  HMI1_DECREMENT_PB_1S  "HMI1 Flow Rate Selector Decrement PB 1-Shot" %
%   N25:80  HMI1_PB_VALUE  "HMI1 Flow Rate Calculator Selection 0 = Manual 1 -> 4 = WY's" %
%   N25:81  HMI_PB_MIN  "HMI Flow Rate Calculator Selection Minimum Value 0" %
%   Q16:1  HMI1_SKIP  "HMI1 Skip to Rung Shown" %
%   N25:82  HMI_PB_MAX  "HMI Flow Rate Calculator Selection Maximum Value -4" %
% Rung: 2 %
% This Rung Provides a
% Destination for the
% HMI1
% Jump to Statement %
SOR LBL Q16:1 MOV N25:80 N25:80 EOR
%   Q16:1  HMI1_SKIP  "HMI1 Skip to Rung Shown" %
%   N25:80  HMI1_PB_VALUE  "HMI1 Flow Rate Calculator Selection 0 = Manual 1 -> 4 = WY's" %

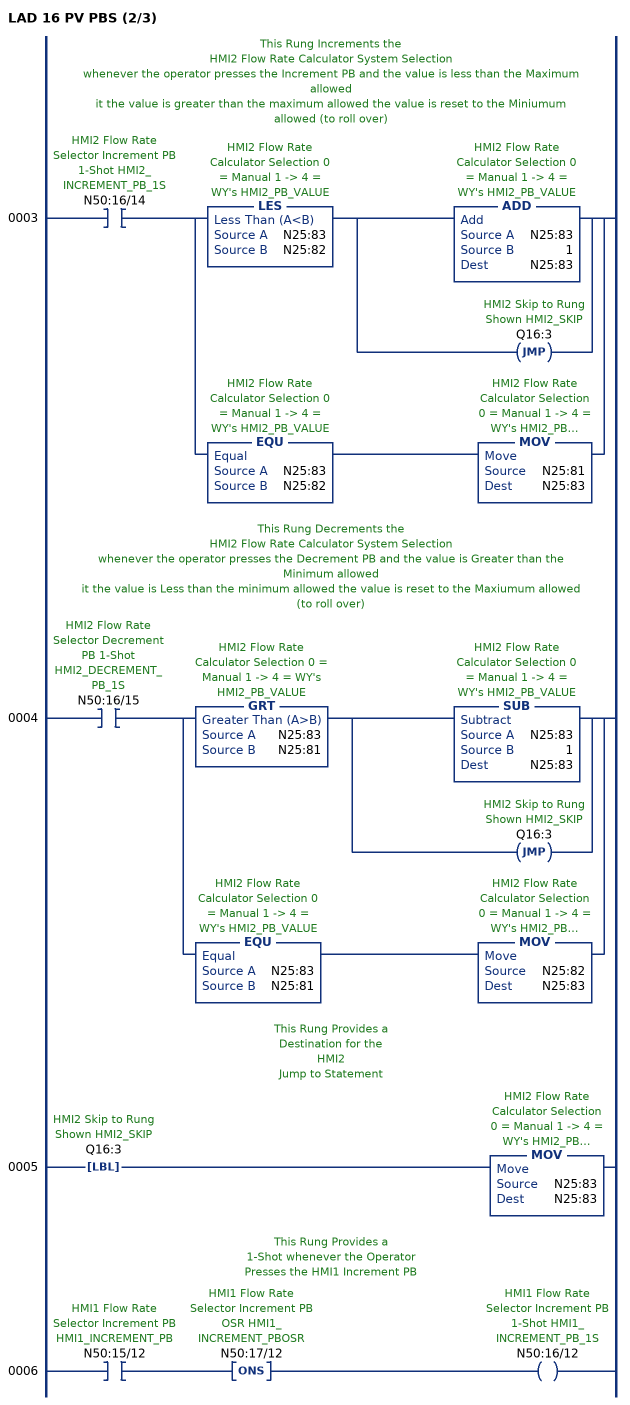
% Rung: 3 %
% This Rung Increments the
% HMI2 Flow Rate Calculator System Selection
% whenever the operator presses the Increment PB and the value is less than the Maximum allowed
% it the value is greater than the maximum allowed the value is reset to the Miniumum allowed (to roll over) %
SOR XIC N50:16/14 BST LES N25:83 N25:82 BST ADD N25:83 1 N25:83 NXB JMP Q16:3 BND NXB EQU N25:83 N25:82 MOV N25:81 N25:83 BND EOR
%   N50:16/14  HMI2_INCREMENT_PB_1S  "HMI2 Flow Rate Selector Increment PB 1-Shot" %
%   N25:83  HMI2_PB_VALUE  "HMI2 Flow Rate Calculator Selection 0 = Manual 1 -> 4 = WY's" %
%   N25:82  HMI_PB_MAX  "HMI Flow Rate Calculator Selection Maximum Value -4" %
%   Q16:3  HMI2_SKIP  "HMI2 Skip to Rung Shown" %
%   N25:81  HMI_PB_MIN  "HMI Flow Rate Calculator Selection Minimum Value 0" %
% Rung: 4 %
% This Rung Decrements the
% HMI2 Flow Rate Calculator System Selection
% whenever the operator presses the Decrement PB and the value is Greater than the Minimum allowed
% it the value is Less than the minimum allowed the value is reset to the Maxiumum allowed (to roll over) %
SOR XIC N50:16/15 BST GRT N25:83 N25:81 BST SUB N25:83 1 N25:83 NXB JMP Q16:3 BND NXB EQU N25:83 N25:81 MOV N25:82 N25:83 BND EOR
%   N50:16/15  HMI2_DECREMENT_PB_1S  "HMI2 Flow Rate Selector Decrement PB 1-Shot" %
%   N25:83  HMI2_PB_VALUE  "HMI2 Flow Rate Calculator Selection 0 = Manual 1 -> 4 = WY's" %
%   N25:81  HMI_PB_MIN  "HMI Flow Rate Calculator Selection Minimum Value 0" %
%   Q16:3  HMI2_SKIP  "HMI2 Skip to Rung Shown" %
%   N25:82  HMI_PB_MAX  "HMI Flow Rate Calculator Selection Maximum Value -4" %
% Rung: 5 %
% This Rung Provides a
% Destination for the
% HMI2
% Jump to Statement %
SOR LBL Q16:3 MOV N25:83 N25:83 EOR
%   Q16:3  HMI2_SKIP  "HMI2 Skip to Rung Shown" %
%   N25:83  HMI2_PB_VALUE  "HMI2 Flow Rate Calculator Selection 0 = Manual 1 -> 4 = WY's" %
% Rung: 6 %
% This Rung Provides a
% 1-Shot whenever the Operator
% Presses the HMI1 Increment PB %
SOR XIC N50:15/12 OSR N50:17/12 OTE N50:16/12 EOR
%   N50:15/12  HMI1_INCREMENT_PB  "HMI1 Flow Rate Selector Increment PB" %
%   N50:17/12  HMI1_INCREMENT_PBOSR  "HMI1 Flow Rate Selector Increment PB OSR" %
%   N50:16/12  HMI1_INCREMENT_PB_1S  "HMI1 Flow Rate Selector Increment PB 1-Shot" %

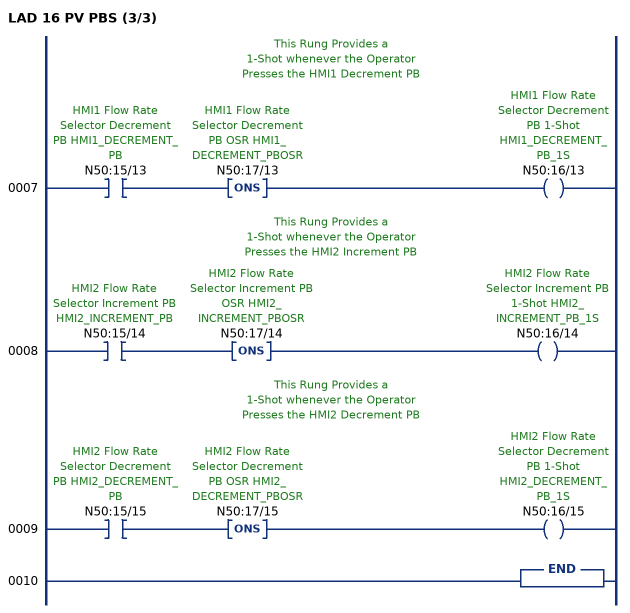
% Rung: 7 %
% This Rung Provides a
% 1-Shot whenever the Operator
% Presses the HMI1 Decrement PB %
SOR XIC N50:15/13 OSR N50:17/13 OTE N50:16/13 EOR
%   N50:15/13  HMI1_DECREMENT_PB  "HMI1 Flow Rate Selector Decrement PB" %
%   N50:17/13  HMI1_DECREMENT_PBOSR  "HMI1 Flow Rate Selector Decrement PB OSR" %
%   N50:16/13  HMI1_DECREMENT_PB_1S  "HMI1 Flow Rate Selector Decrement PB 1-Shot" %
% Rung: 8 %
% This Rung Provides a
% 1-Shot whenever the Operator
% Presses the HMI2 Increment PB %
SOR XIC N50:15/14 OSR N50:17/14 OTE N50:16/14 EOR
%   N50:15/14  HMI2_INCREMENT_PB  "HMI2 Flow Rate Selector Increment PB" %
%   N50:17/14  HMI2_INCREMENT_PBOSR  "HMI2 Flow Rate Selector Increment PB OSR" %
%   N50:16/14  HMI2_INCREMENT_PB_1S  "HMI2 Flow Rate Selector Increment PB 1-Shot" %
% Rung: 9 %
% This Rung Provides a
% 1-Shot whenever the Operator
% Presses the HMI2 Decrement PB %
SOR XIC N50:15/15 OSR N50:17/15 OTE N50:16/15 EOR
%   N50:15/15  HMI2_DECREMENT_PB  "HMI2 Flow Rate Selector Decrement PB" %
%   N50:17/15  HMI2_DECREMENT_PBOSR  "HMI2 Flow Rate Selector Decrement PB OSR" %
%   N50:16/15  HMI2_DECREMENT_PB_1S  "HMI2 Flow Rate Selector Decrement PB 1-Shot" %
% Rung: 10 %
SOR END EOR

LADDER 17 "VFD USERS"    % Determines which user is using each VFD %
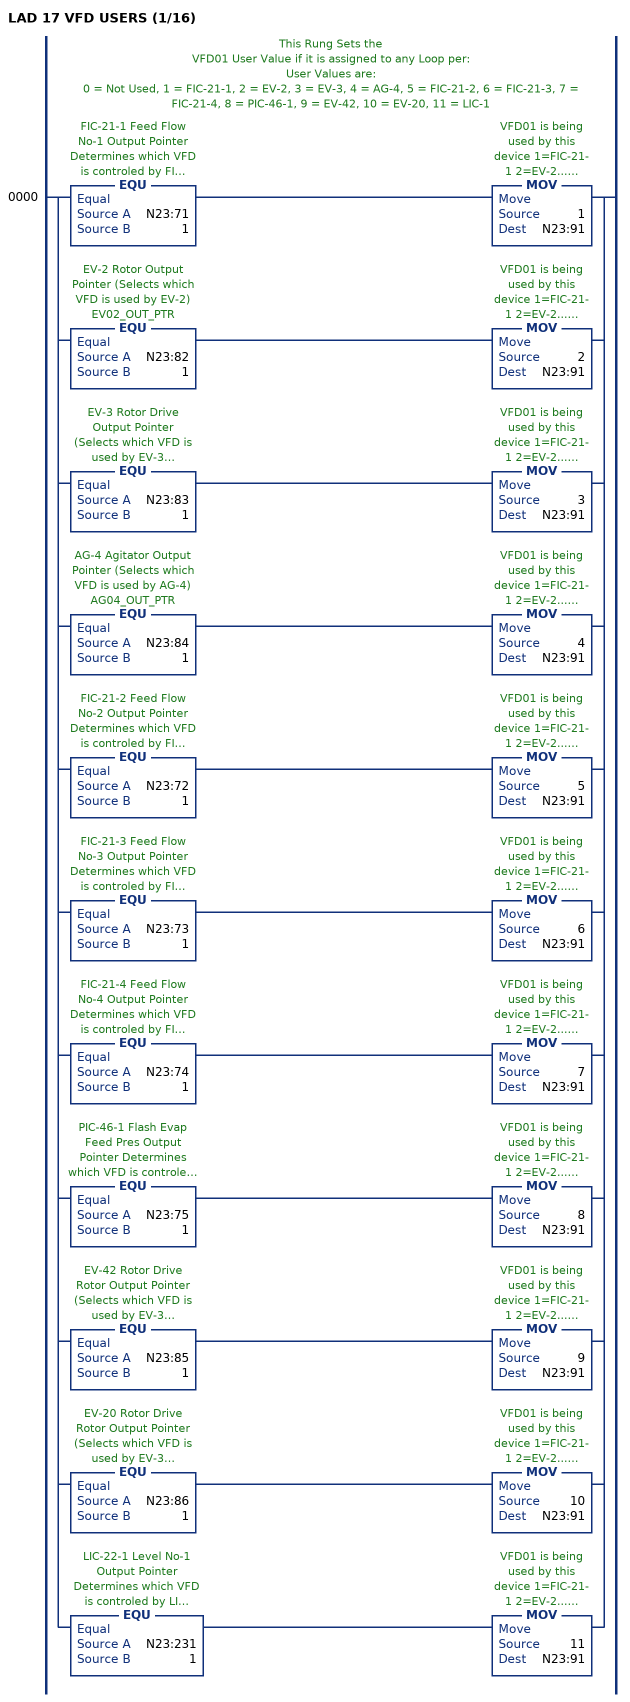
% Rung: 0 %
% This Rung Sets the
% VFD01 User Value if it is assigned to any Loop per:
% 
% User Values are:
% 0 = Not Used, 1 = FIC-21-1, 2 = EV-2, 3 = EV-3, 4 = AG-4, 5 = FIC-21-2, 6 = FIC-21-3, 7 = FIC-21-4, 8 = PIC-46-1, 9 = EV-42, 10 = EV-20, 11 = LIC-1 %
SOR BST EQU N23:71 1 MOV 1 N23:91 NXB EQU N23:82 1 MOV 2 N23:91 NXB EQU N23:83 1 MOV 3 N23:91 NXB EQU N23:84 1 MOV 4 N23:91 NXB EQU N23:72 1 MOV 5 N23:91 NXB EQU N23:73 1 MOV 6 N23:91 NXB EQU N23:74 1 MOV 7 N23:91 NXB EQU N23:75 1 MOV 8 N23:91 NXB EQU N23:85 1 MOV 9 N23:91 NXB EQU N23:86 1 MOV 10 N23:91 NXB EQU N23:231 1 MOV 11 N23:91 BND EOR
%   N23:71  FIC211_OUT_PTR  "FIC-21-1 Feed Flow No-1 Output Pointer Determines which VFD is controled by FIC" %
%   N23:91  VFD01_USER  "VFD01 is being used by this device 1=FIC-21-1 2=EV-2...." %
%   N23:82  EV02_OUT_PTR  "EV-2 Rotor Output Pointer (Selects which VFD is used by EV-2)" %
%   N23:83  EV03_OUT_PTR  "EV-3 Rotor Drive Output Pointer (Selects which VFD is used by EV-3)" %
%   N23:84  AG04_OUT_PTR  "AG-4 Agitator Output Pointer (Selects which VFD is used by AG-4)" %
%   N23:72  FIC212_OUT_PTR  "FIC-21-2 Feed Flow No-2 Output Pointer Determines which VFD is controled by FIC" %
%   N23:73  FIC213_OUT_PTR  "FIC-21-3 Feed Flow No-3 Output Pointer Determines which VFD is controled by FIC" %
%   N23:74  FIC214_OUT_PTR  "FIC-21-4 Feed Flow No-4 Output Pointer Determines which VFD is controled by FIC" %
%   N23:75  PIC461_OUT_PTR  "PIC-46-1 Flash Evap Feed Pres Output Pointer Determines which VFD is controled by FIC" %
%   N23:85  EV42_OUT_PTR  "EV-42 Rotor Drive Rotor Output Pointer (Selects which VFD is used by EV-3)" %
%   N23:86  EV20_OUT_PTR  "EV-20 Rotor Drive Rotor Output Pointer (Selects which VFD is used by EV-3)" %
%   N23:231  LIC221_OUT_PTR  "LIC-22-1 Level No-1 Output Pointer Determines which VFD is controled by LIC" %

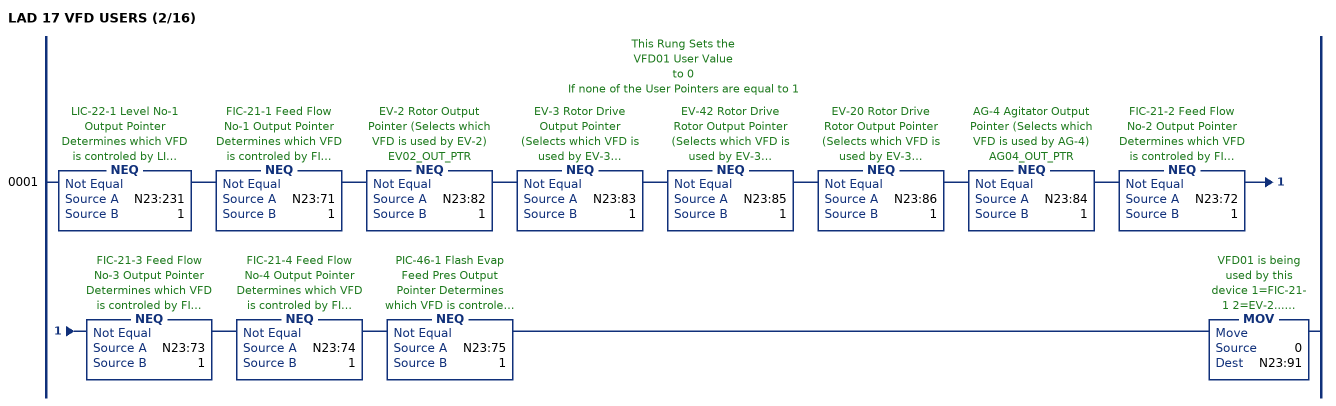
% Rung: 1 %
% This Rung Sets the
% VFD01 User Value
% to 0
% If none of the User Pointers are equal to 1 %
SOR NEQ N23:231 1 NEQ N23:71 1 NEQ N23:82 1 NEQ N23:83 1 NEQ N23:85 1 NEQ N23:86 1 NEQ N23:84 1 NEQ N23:72 1 NEQ N23:73 1 NEQ N23:74 1 NEQ N23:75 1 MOV 0 N23:91 EOR
%   N23:231  LIC221_OUT_PTR  "LIC-22-1 Level No-1 Output Pointer Determines which VFD is controled by LIC" %
%   N23:71  FIC211_OUT_PTR  "FIC-21-1 Feed Flow No-1 Output Pointer Determines which VFD is controled by FIC" %
%   N23:82  EV02_OUT_PTR  "EV-2 Rotor Output Pointer (Selects which VFD is used by EV-2)" %
%   N23:83  EV03_OUT_PTR  "EV-3 Rotor Drive Output Pointer (Selects which VFD is used by EV-3)" %
%   N23:85  EV42_OUT_PTR  "EV-42 Rotor Drive Rotor Output Pointer (Selects which VFD is used by EV-3)" %
%   N23:86  EV20_OUT_PTR  "EV-20 Rotor Drive Rotor Output Pointer (Selects which VFD is used by EV-3)" %
%   N23:84  AG04_OUT_PTR  "AG-4 Agitator Output Pointer (Selects which VFD is used by AG-4)" %
%   N23:72  FIC212_OUT_PTR  "FIC-21-2 Feed Flow No-2 Output Pointer Determines which VFD is controled by FIC" %
%   N23:73  FIC213_OUT_PTR  "FIC-21-3 Feed Flow No-3 Output Pointer Determines which VFD is controled by FIC" %
%   N23:74  FIC214_OUT_PTR  "FIC-21-4 Feed Flow No-4 Output Pointer Determines which VFD is controled by FIC" %
%   N23:75  PIC461_OUT_PTR  "PIC-46-1 Flash Evap Feed Pres Output Pointer Determines which VFD is controled by FIC" %
%   N23:91  VFD01_USER  "VFD01 is being used by this device 1=FIC-21-1 2=EV-2...." %

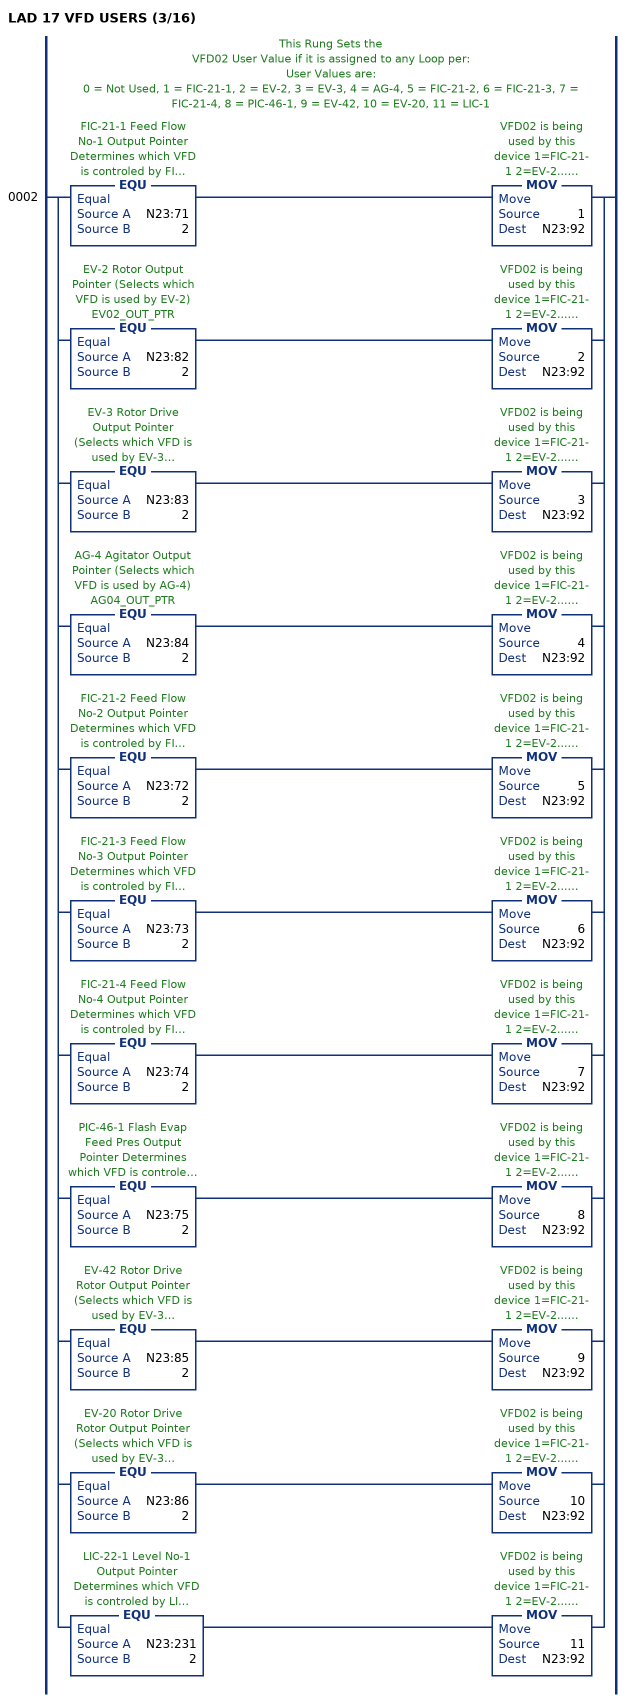
% Rung: 2 %
% This Rung Sets the
% VFD02 User Value if it is assigned to any Loop per:
% 
% User Values are:
% 0 = Not Used, 1 = FIC-21-1, 2 = EV-2, 3 = EV-3, 4 = AG-4, 5 = FIC-21-2, 6 = FIC-21-3, 7 = FIC-21-4, 8 = PIC-46-1, 9 = EV-42, 10 = EV-20, 11 = LIC-1 %
SOR BST EQU N23:71 2 MOV 1 N23:92 NXB EQU N23:82 2 MOV 2 N23:92 NXB EQU N23:83 2 MOV 3 N23:92 NXB EQU N23:84 2 MOV 4 N23:92 NXB EQU N23:72 2 MOV 5 N23:92 NXB EQU N23:73 2 MOV 6 N23:92 NXB EQU N23:74 2 MOV 7 N23:92 NXB EQU N23:75 2 MOV 8 N23:92 NXB EQU N23:85 2 MOV 9 N23:92 NXB EQU N23:86 2 MOV 10 N23:92 NXB EQU N23:231 2 MOV 11 N23:92 BND EOR
%   N23:71  FIC211_OUT_PTR  "FIC-21-1 Feed Flow No-1 Output Pointer Determines which VFD is controled by FIC" %
%   N23:92  VFD02_USER  "VFD02 is being used by this device 1=FIC-21-1 2=EV-2...." %
%   N23:82  EV02_OUT_PTR  "EV-2 Rotor Output Pointer (Selects which VFD is used by EV-2)" %
%   N23:83  EV03_OUT_PTR  "EV-3 Rotor Drive Output Pointer (Selects which VFD is used by EV-3)" %
%   N23:84  AG04_OUT_PTR  "AG-4 Agitator Output Pointer (Selects which VFD is used by AG-4)" %
%   N23:72  FIC212_OUT_PTR  "FIC-21-2 Feed Flow No-2 Output Pointer Determines which VFD is controled by FIC" %
%   N23:73  FIC213_OUT_PTR  "FIC-21-3 Feed Flow No-3 Output Pointer Determines which VFD is controled by FIC" %
%   N23:74  FIC214_OUT_PTR  "FIC-21-4 Feed Flow No-4 Output Pointer Determines which VFD is controled by FIC" %
%   N23:75  PIC461_OUT_PTR  "PIC-46-1 Flash Evap Feed Pres Output Pointer Determines which VFD is controled by FIC" %
%   N23:85  EV42_OUT_PTR  "EV-42 Rotor Drive Rotor Output Pointer (Selects which VFD is used by EV-3)" %
%   N23:86  EV20_OUT_PTR  "EV-20 Rotor Drive Rotor Output Pointer (Selects which VFD is used by EV-3)" %
%   N23:231  LIC221_OUT_PTR  "LIC-22-1 Level No-1 Output Pointer Determines which VFD is controled by LIC" %

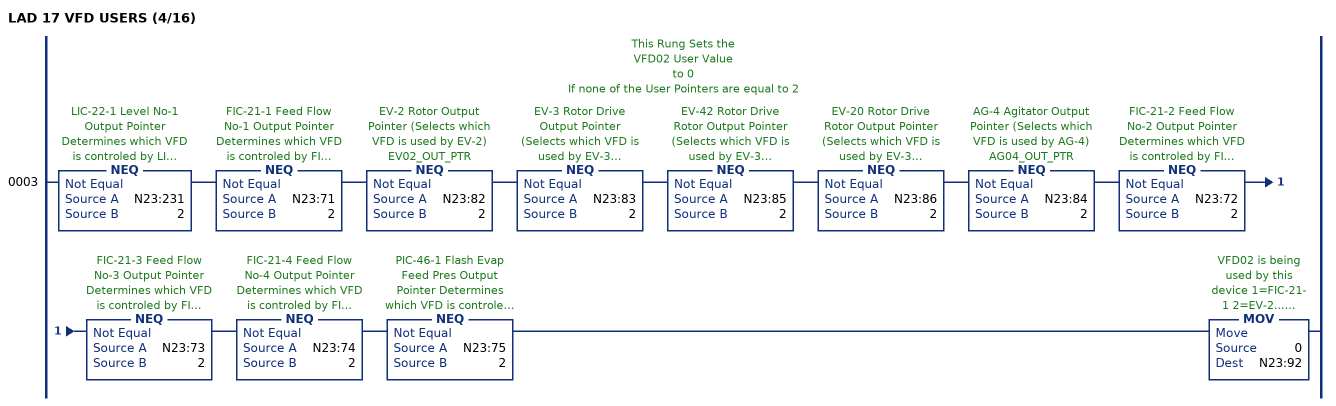
% Rung: 3 %
% This Rung Sets the
% VFD02 User Value
% to 0
% If none of the User Pointers are equal to 2 %
SOR NEQ N23:231 2 NEQ N23:71 2 NEQ N23:82 2 NEQ N23:83 2 NEQ N23:85 2 NEQ N23:86 2 NEQ N23:84 2 NEQ N23:72 2 NEQ N23:73 2 NEQ N23:74 2 NEQ N23:75 2 MOV 0 N23:92 EOR
%   N23:231  LIC221_OUT_PTR  "LIC-22-1 Level No-1 Output Pointer Determines which VFD is controled by LIC" %
%   N23:71  FIC211_OUT_PTR  "FIC-21-1 Feed Flow No-1 Output Pointer Determines which VFD is controled by FIC" %
%   N23:82  EV02_OUT_PTR  "EV-2 Rotor Output Pointer (Selects which VFD is used by EV-2)" %
%   N23:83  EV03_OUT_PTR  "EV-3 Rotor Drive Output Pointer (Selects which VFD is used by EV-3)" %
%   N23:85  EV42_OUT_PTR  "EV-42 Rotor Drive Rotor Output Pointer (Selects which VFD is used by EV-3)" %
%   N23:86  EV20_OUT_PTR  "EV-20 Rotor Drive Rotor Output Pointer (Selects which VFD is used by EV-3)" %
%   N23:84  AG04_OUT_PTR  "AG-4 Agitator Output Pointer (Selects which VFD is used by AG-4)" %
%   N23:72  FIC212_OUT_PTR  "FIC-21-2 Feed Flow No-2 Output Pointer Determines which VFD is controled by FIC" %
%   N23:73  FIC213_OUT_PTR  "FIC-21-3 Feed Flow No-3 Output Pointer Determines which VFD is controled by FIC" %
%   N23:74  FIC214_OUT_PTR  "FIC-21-4 Feed Flow No-4 Output Pointer Determines which VFD is controled by FIC" %
%   N23:75  PIC461_OUT_PTR  "PIC-46-1 Flash Evap Feed Pres Output Pointer Determines which VFD is controled by FIC" %
%   N23:92  VFD02_USER  "VFD02 is being used by this device 1=FIC-21-1 2=EV-2...." %

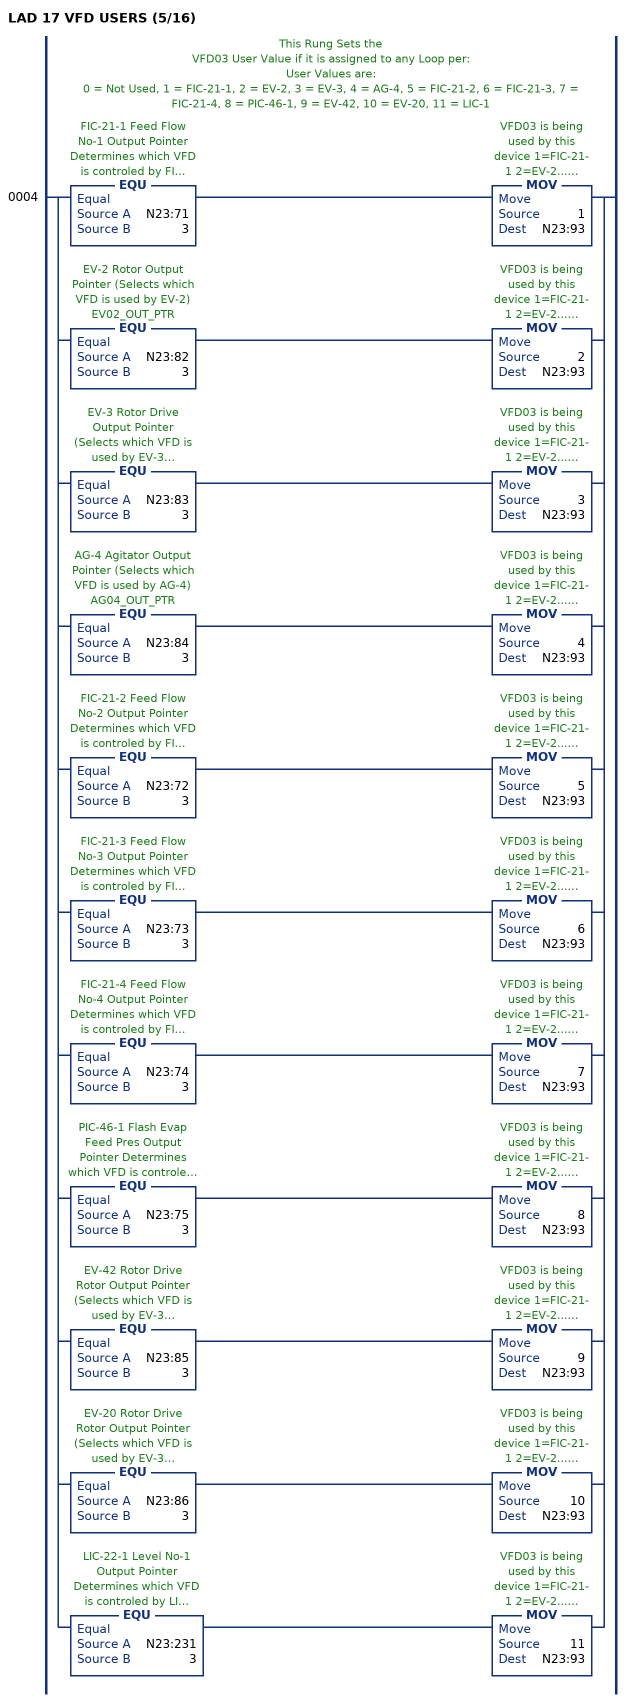
% Rung: 4 %
% This Rung Sets the
% VFD03 User Value if it is assigned to any Loop per:
% 
% User Values are:
% 0 = Not Used, 1 = FIC-21-1, 2 = EV-2, 3 = EV-3, 4 = AG-4, 5 = FIC-21-2, 6 = FIC-21-3, 7 = FIC-21-4, 8 = PIC-46-1, 9 = EV-42, 10 = EV-20, 11 = LIC-1 %
SOR BST EQU N23:71 3 MOV 1 N23:93 NXB EQU N23:82 3 MOV 2 N23:93 NXB EQU N23:83 3 MOV 3 N23:93 NXB EQU N23:84 3 MOV 4 N23:93 NXB EQU N23:72 3 MOV 5 N23:93 NXB EQU N23:73 3 MOV 6 N23:93 NXB EQU N23:74 3 MOV 7 N23:93 NXB EQU N23:75 3 MOV 8 N23:93 NXB EQU N23:85 3 MOV 9 N23:93 NXB EQU N23:86 3 MOV 10 N23:93 NXB EQU N23:231 3 MOV 11 N23:93 BND EOR
%   N23:71  FIC211_OUT_PTR  "FIC-21-1 Feed Flow No-1 Output Pointer Determines which VFD is controled by FIC" %
%   N23:93  VFD03_USER  "VFD03 is being used by this device 1=FIC-21-1 2=EV-2...." %
%   N23:82  EV02_OUT_PTR  "EV-2 Rotor Output Pointer (Selects which VFD is used by EV-2)" %
%   N23:83  EV03_OUT_PTR  "EV-3 Rotor Drive Output Pointer (Selects which VFD is used by EV-3)" %
%   N23:84  AG04_OUT_PTR  "AG-4 Agitator Output Pointer (Selects which VFD is used by AG-4)" %
%   N23:72  FIC212_OUT_PTR  "FIC-21-2 Feed Flow No-2 Output Pointer Determines which VFD is controled by FIC" %
%   N23:73  FIC213_OUT_PTR  "FIC-21-3 Feed Flow No-3 Output Pointer Determines which VFD is controled by FIC" %
%   N23:74  FIC214_OUT_PTR  "FIC-21-4 Feed Flow No-4 Output Pointer Determines which VFD is controled by FIC" %
%   N23:75  PIC461_OUT_PTR  "PIC-46-1 Flash Evap Feed Pres Output Pointer Determines which VFD is controled by FIC" %
%   N23:85  EV42_OUT_PTR  "EV-42 Rotor Drive Rotor Output Pointer (Selects which VFD is used by EV-3)" %
%   N23:86  EV20_OUT_PTR  "EV-20 Rotor Drive Rotor Output Pointer (Selects which VFD is used by EV-3)" %
%   N23:231  LIC221_OUT_PTR  "LIC-22-1 Level No-1 Output Pointer Determines which VFD is controled by LIC" %

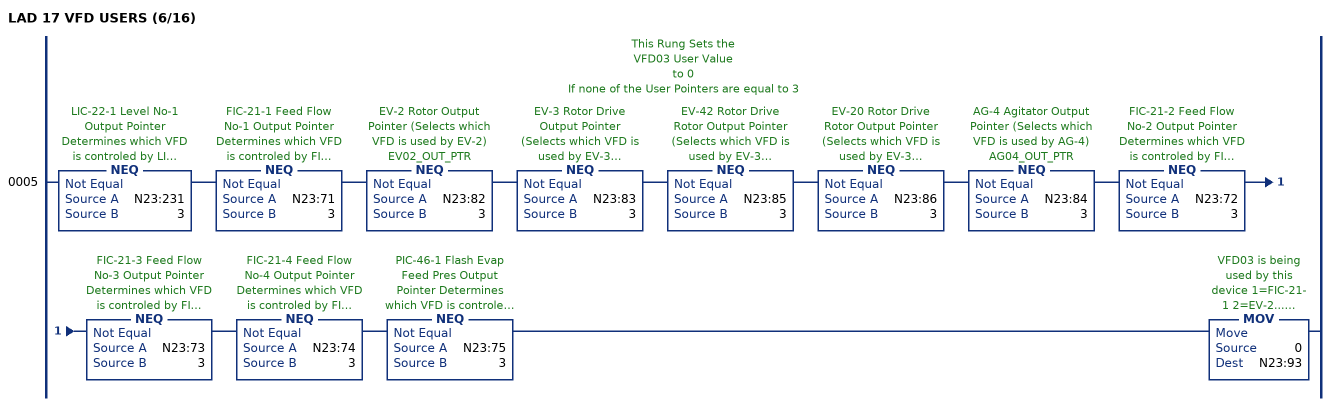
% Rung: 5 %
% This Rung Sets the
% VFD03 User Value
% to 0
% If none of the User Pointers are equal to 3 %
SOR NEQ N23:231 3 NEQ N23:71 3 NEQ N23:82 3 NEQ N23:83 3 NEQ N23:85 3 NEQ N23:86 3 NEQ N23:84 3 NEQ N23:72 3 NEQ N23:73 3 NEQ N23:74 3 NEQ N23:75 3 MOV 0 N23:93 EOR
%   N23:231  LIC221_OUT_PTR  "LIC-22-1 Level No-1 Output Pointer Determines which VFD is controled by LIC" %
%   N23:71  FIC211_OUT_PTR  "FIC-21-1 Feed Flow No-1 Output Pointer Determines which VFD is controled by FIC" %
%   N23:82  EV02_OUT_PTR  "EV-2 Rotor Output Pointer (Selects which VFD is used by EV-2)" %
%   N23:83  EV03_OUT_PTR  "EV-3 Rotor Drive Output Pointer (Selects which VFD is used by EV-3)" %
%   N23:85  EV42_OUT_PTR  "EV-42 Rotor Drive Rotor Output Pointer (Selects which VFD is used by EV-3)" %
%   N23:86  EV20_OUT_PTR  "EV-20 Rotor Drive Rotor Output Pointer (Selects which VFD is used by EV-3)" %
%   N23:84  AG04_OUT_PTR  "AG-4 Agitator Output Pointer (Selects which VFD is used by AG-4)" %
%   N23:72  FIC212_OUT_PTR  "FIC-21-2 Feed Flow No-2 Output Pointer Determines which VFD is controled by FIC" %
%   N23:73  FIC213_OUT_PTR  "FIC-21-3 Feed Flow No-3 Output Pointer Determines which VFD is controled by FIC" %
%   N23:74  FIC214_OUT_PTR  "FIC-21-4 Feed Flow No-4 Output Pointer Determines which VFD is controled by FIC" %
%   N23:75  PIC461_OUT_PTR  "PIC-46-1 Flash Evap Feed Pres Output Pointer Determines which VFD is controled by FIC" %
%   N23:93  VFD03_USER  "VFD03 is being used by this device 1=FIC-21-1 2=EV-2...." %

